(* Stop *)
	IF xStop THEN
		(* init. FB vel / abs / rel *)
		xMoveVel:=FALSE;
		xMoveRel:=FALSE;
		xMoveAbs:=FALSE;
		xMoveModulo:=FALSE;
		xNewVelocity:=FALSE;
		xNewPosition:=FALSE;
		xStartTimerComm:=FALSE;
		xHoming:=FALSE;
		IF (iTmpFctNr <> 19) THEN
			xCalcAngleRefIndex:=FALSE;
		END_IF;
		(* flag oscillation off *)
		xOscillation:=FALSE;
		(* FB stop *)
		xStopAxisVelCtrlActive:=FALSE;
		IF (T_Axis.T_Config_Gen.iTyp <> 1) THEN
			fbAxisStop(	Execute:=TRUE,
						Deceleration:=T_Axis.T_CtrleSingle.lrDecceleration,
						Jerk:=T_Axis.T_CtrleSingle.lrJerk,
						Axis:=T_AxisRefIn);
		ELSE
			IF NOT(gxZAxisVelocityCtrlActive) THEN
				fbAxisStop(	Execute:=TRUE,
							Deceleration:=T_Axis.T_CtrleSingle.lrDecceleration,
							Jerk:=T_Axis.T_CtrleSingle.lrJerk,
							Axis:=T_AxisRefIn);
			ELSE
				xStopAxisVelCtrlActive:=TRUE;
			END_IF;
		END_IF;
		(* select bit not moving *)
		dwTmp:=T_Axis.T_LiveValue.dwState AND 16#4;
		IF NOT(xStopAxisVelCtrlActive) THEN
			IF (fbAxisStop.Done AND dwTmp = 16#4) OR fbAxisStop.Error THEN
				IF fbAxisStop.Error OR (NOT(xResetAxis) AND NOT(xResetAX5000Axis) AND NOT(xCalcAngleRefIndex) )THEN
					xResetAxis:=xCalcAngleRefIndex:=xResetAX5000Axis:=FALSE;
				(* confirm reset if error activ or if reset is not activ *)
					T_Axis.T_CtrleSingle.xDone:=fbAxisStop.Done;
					T_Axis.T_CtrleSingle.xErr:= fbAxisStop.Error;
					T_Axis.T_CtrleSingle.udiErrorID:=fbAxisStop.ErrorID;
					(* desactiv reset axis *)
					IF xResetAxis THEN xResetAxis:=FALSE; END_IF
					IF (T_Axis.T_Config_Gen.iTyp = 1) AND gxZFollowDistanceError THEN
						T_Axis.T_CtrleSingle.xDone:=FALSE;
						T_Axis.T_CtrleSingle.xErr:= TRUE;
						T_Axis.T_CtrleSingle.udiErrorID:=16#4550;	(* Schleppabstandsfehler *)
					END_IF;
				END_IF
				(* flag stop off *)
				xStop:=FALSE;
				tTimeCommLeft1:=TimerCommTimeLeft1.ET;
				xStartTimerComm1:=FALSE;
				(* reset flag busy *)
				T_Axis.T_CtrleSingle.xBusyNewPosAndVel:=FALSE;
				(* Init. Stop FB *)
				fbAxisStop(Execute:=FALSE, Axis:=T_AxisRefIn);
				IF xActiveFollowError AND NOT(fbAxisStop.Error) THEN
					T_Axis.T_CtrleSingle.xDone:=FALSE;
					T_Axis.T_CtrleSingle.xErr:= FALSE;
					T_Axis.T_CtrleSingle.udiErrorID:=0;
					xActiveFollowError:=FALSE;
					iStepResetFB:=1;
					xResetAxis:=TRUE;
					RETURN;
				END_IF;
				IF gxSpindleOverloadError AND (T_Axis.T_Config_Gen.iTyp = 2) THEN
					gxSpindleOverloadError:=FALSE;
					T_Axis.T_CtrleSingle.xDone:=FALSE;
					T_Axis.T_CtrleSingle.xErr:= TRUE;
					T_Axis.T_CtrleSingle.udiErrorID:=16#F502;
				END_IF;
			END_IF
		ELSE
			CASE iStopAxis OF
			1:	TONWaitStop(IN:=FALSE);
				iStepResetFB:=1;
				xResetAxis:=TRUE;
				iStopAxis:=iStopAxis + 1;
			2:	IF NOT(xResetAxis) THEN
					iStopAxis:=iStopAxis + 1;
				END_IF;
			3:	TONWaitStop(IN:=TRUE,PT:=T#0.3s);
				IF TONWaitStop.Q THEN
					TONWaitStop(IN:=FALSE);
					T_Axis.T_CtrleSingle.xDone:=TRUE;
					T_Axis.T_CtrleSingle.xErr:= FALSE;
					T_Axis.T_CtrleSingle.udiErrorID:=16#0;
					xStop:=FALSE;
					xStopAxisVelCtrlActive:=FALSE;
					iStopAxis:=1;
					IF (T_Axis.T_Config_Gen.iTyp = 1) AND gxZFollowDistanceError THEN
						T_Axis.T_CtrleSingle.xDone:=FALSE;
						T_Axis.T_CtrleSingle.xErr:= TRUE;
						T_Axis.T_CtrleSingle.udiErrorID:=16#4550;	(* Schleppabstandsfehler *)
					END_IF;
				END_IF;
			END_CASE;
		END_IF;
	ELSE fbAxisStop(Execute:=FALSE, Axis:=T_AxisRefIn); END_IF

(* Velocity *)
	IF xMoveVel AND NOT(fbAxisMoveVelocity.InVelocity) THEN
		IF T_Axis.T_CtrleSingle.lrVelocity >= 0 THEN
		(* positiv direction =1*)
			iDirectionVel:=MC_Positive_Direction;
		ELSE
		(* negativ direction =3*)
			iDirectionVel:=MC_Negative_Direction;
		END_IF
		IF (T_Axis.T_Config_Gen.iTyp <> 2) THEN
			rVelocity:=ABS(lrOverrideVel);
		ELSE
			rVelocity:=ABS(lrOverrideVel) * T_Axis.T_CtrleSingle.lrScaleFactor;
		END_IF;
		fbAxisMoveVelocity(	Execute:=TRUE,
							Velocity:=rVelocity,
							Acceleration:=T_Axis.T_CtrleSingle.lrAcceleration,
							Deceleration:=T_Axis.T_CtrleSingle.lrDecceleration,
							Jerk:=T_Axis.T_CtrleSingle.lrJerk,
							Direction:=iDirectionVel,
							Axis:=T_AxisRefIn);
		IF fbAxisMoveVelocity.InVelocity OR fbAxisMoveVelocity.Error THEN
			T_Axis.T_CtrleSingle.xDone:=fbAxisMoveVelocity.InVelocity;
			T_Axis.T_CtrleSingle.xErr:= fbAxisMoveVelocity.Error;
			T_Axis.T_CtrleSingle.udiErrorID:=fbAxisMoveVelocity.ErrorID;
			(* flag velocity off *)
			xMoveVel:=FALSE;
			(* Init. FB Move *)
			fbAxisMoveVelocity(Execute:=FALSE, Axis:=T_AxisRefIn);
		END_IF
	ELSE fbAxisMoveVelocity(Execute:=FALSE, Axis:=T_AxisRefIn); END_IF

(* Move absolute *)
	IF xMoveAbs THEN
		fbAxisMoveAbsolute(	Execute:=TRUE,
							Position:=T_Axis.T_CtrleSingle.lrPosition,
							Velocity:=ABS(lrOverrideVel),
							Acceleration:=T_Axis.T_CtrleSingle.lrAcceleration,
							Deceleration:=T_Axis.T_CtrleSingle.lrDecceleration,
							Jerk:=T_Axis.T_CtrleSingle.lrJerk,
							Axis:=T_AxisRefIn);
		IF fbAxisMoveAbsolute.Done OR fbAxisMoveAbsolute.Error THEN
			IF NOT(xCalcAngleRefIndex) OR fbAxisMoveAbsolute.Error THEN
				xCalcAngleRefIndex:=FALSE;
				IF NOT(T_Axis.T_CtrleSingle.xErr) THEN	(* xNewVelocity könnte einen Fehler generiert haben, aber diese Funktion ist noch aktiv und darf daher nicht überschrieben werden *)
					T_Axis.T_CtrleSingle.xDone:=fbAxisMoveAbsolute.Done;
					T_Axis.T_CtrleSingle.xErr:= fbAxisMoveAbsolute.Error;
					T_Axis.T_CtrleSingle.udiErrorID:=fbAxisMoveAbsolute.ErrorID;
				END_IF;
				(* test if move has been stopped *)
				IF fbAxisMoveAbsolute.ErrorID = 16#4B00 THEN
				(* clear error *)
					T_Axis.T_CtrleSingle.xDone:=TRUE;
					T_Axis.T_CtrleSingle.xErr:= FALSE;
					T_Axis.T_CtrleSingle.udiErrorID:=16#0;
				END_IF
			END_IF;
			(* flag move absolute off *)
			xMoveAbs:=FALSE;
			(* init. FB *)
			fbAxisMoveAbsolute(Execute:=FALSE, Axis:=T_AxisRefIn);
		END_IF
	ELSE fbAxisMoveAbsolute(Execute:=FALSE, Axis:=T_AxisRefIn); END_IF

(* Move relative *)
	IF xMoveRel THEN
		IF (T_Axis.T_Config_Gen.iTyp <> 2) THEN
			lrDistance:=T_Axis.T_CtrleSingle.lrDistance;
		ELSE
			CASE T_ExchgParam.bToolSpindleActive OF
			1:	(* Maxon Spindel *)
				lrDistance:=T_Axis.T_CtrleSingle.lrDistance / grScaleSAxis_Distance_SM;
			2,3:	(* Beckhoff Spindel *)
				lrDistance:=T_Axis.T_CtrleSingle.lrDistance / grScaleSAxis_Distance_L;
			END_CASE;
		END_IF;
		fbAxisMoveRelative(	Execute:=TRUE,
							Distance:=lrDistance,
							Velocity:=lrOverrideVel,
							Acceleration:=T_Axis.T_CtrleSingle.lrAcceleration,
							Deceleration:=T_Axis.T_CtrleSingle.lrDecceleration,
							Jerk:=T_Axis.T_CtrleSingle.lrJerk,
							Axis:=T_AxisRefIn);
		IF fbAxisMoveRelative.Done OR fbAxisMoveRelative.Error THEN
			IF (NOT(xOscillation) AND NOT(xCalcAngleRefIndex)) OR fbAxisMoveRelative.Error THEN
				xOscillation:=xCalcAngleRefIndex:=FALSE;
			(* normal control variable settings if oscillation disable *)
				IF NOT(T_Axis.T_CtrleSingle.xErr) THEN	(* xNewVelocity könnte einen Fehler generiert haben, aber diese Funktion ist noch aktiv und darf daher nicht überschrieben werden *)
					T_Axis.T_CtrleSingle.xDone:=fbAxisMoveRelative.Done;
					T_Axis.T_CtrleSingle.xErr:= fbAxisMoveRelative.Error;
					T_Axis.T_CtrleSingle.udiErrorID:=fbAxisMoveRelative.ErrorID;
				END_IF;
				(* test if move has been stopped *)
				IF fbAxisMoveRelative.ErrorID = 16#4B00 THEN
				(* clear error *)
					T_Axis.T_CtrleSingle.xDone:=TRUE;
					T_Axis.T_CtrleSingle.xErr:= FALSE;
					T_Axis.T_CtrleSingle.udiErrorID:=16#0;
				END_IF
			END_IF
			(* flag move relative off *)
			xMoveRel:=FALSE;
			(* init. FB *)
			fbAxisMoveRelative(Execute:=FALSE, Axis:=T_AxisRefIn);
		END_IF
	ELSE fbAxisMoveRelative(Execute:=FALSE, Axis:=T_AxisRefIn); END_IF

(* Move modulo *)
	IF xMoveModulo THEN
		fbAxisMoveModulo(	Execute:= TRUE,
							Position:= T_Axis.T_CtrleSingle.lrPosition,
							Velocity:= ABS(lrOverrideVel),
							Acceleration:= T_Axis.T_CtrleSingle.lrAcceleration,
							Deceleration:= T_Axis.T_CtrleSingle.lrDecceleration,
							Jerk:= T_Axis.T_CtrleSingle.lrJerk,
							Direction:= T_Axis.T_CtrleSingle.iModuloDirection,
							Axis:= T_AxisRefIn);
		IF fbAxisMoveModulo.Done OR fbAxisMoveModulo.Error THEN
			xCalcAngleRefIndex:=FALSE;
			T_Axis.T_CtrleSingle.xDone:=fbAxisMoveModulo.Done;
			T_Axis.T_CtrleSingle.xErr:= fbAxisMoveModulo.Error;
			T_Axis.T_CtrleSingle.udiErrorID:=fbAxisMoveModulo.ErrorID;
			(* test if move has been stopped *)
			IF fbAxisMoveModulo.ErrorID = 16#4B00 THEN
			(* clear error *)
				T_Axis.T_CtrleSingle.xDone:=TRUE;
				T_Axis.T_CtrleSingle.xErr:= FALSE;
				T_Axis.T_CtrleSingle.udiErrorID:=16#0;
			END_IF
			(* flag move absolute off *)
			xMoveModulo:=FALSE;
			(* init. FB *)
			fbAxisMoveModulo(Execute:=FALSE, Axis:=T_AxisRefIn);
		END_IF
	ELSE fbAxisMoveModulo(Execute:=FALSE, Axis:=T_AxisRefIn); END_IF

(* Homing *)
	IF xHoming THEN
		IF(T_Axis.T_Config_Gen.iTyp=1) THEN
			lrSetPosition:=T_Axis.T_CtrleSingle.rSetPosition + lrNullPointOffset;
		ELSE
			lrSetPosition:=T_Axis.T_CtrleSingle.rSetPosition;
		END_IF;
		fbAxisHoming(	Execute:=TRUE,
						Position:=lrSetPosition,
						bCalibrationCam:=xRefHoming,
						Axis:=T_AxisRefIn,
						AxisOut:=T_AxisRefOut);
		IF fbAxisHoming.Done OR fbAxisHoming.Error THEN
			IF NOT(xCalcAngleRefIndex) OR fbAxisHoming.Error THEN
				xCalcAngleRefIndex:=FALSE;
				T_Axis.T_CtrleSingle.xDone:=fbAxisHoming.Done;
				T_Axis.T_CtrleSingle.xErr:= fbAxisHoming.Error;
				T_Axis.T_CtrleSingle.udiErrorID:=fbAxisHoming.ErrorID;
			END_IF;
			(* flag homing off *)
			xHoming:=FALSE;
			(* Init. FB Homing *)
			fbAxisHoming(	Execute:=FALSE,
							Axis:=T_AxisRefIn,
							AxisOut:=T_AxisRefOut);
		END_IF
	ELSE
		fbAxisHoming(	Execute:=FALSE,
						Axis:=T_AxisRefIn,
						AxisOut:=T_AxisRefOut);
	END_IF

(* Set override *)
	IF xOverride THEN
		fbAxisSetOverride(Execute:=TRUE,
						Override:=T_Axis.T_CtrleSingle.dwOverride,
						AxisRefIn:=T_AxisRefIn,
						AxisRefOut:=T_AxisRefOut);
		IF fbAxisSetOverride.Done OR fbAxisSetOverride.Error THEN
			T_Axis.T_CtrleSingle.xDone:=fbAxisSetOverride.Done;
			T_Axis.T_CtrleSingle.xErr:= fbAxisSetOverride.Error;
			T_Axis.T_CtrleSingle.udiErrorID:=fbAxisSetOverride.ErrorID;
			(* flag override off *)
			xOverride:=FALSE;
			(* Init. FB Override *)
			fbAxisSetOverride(Execute:=FALSE,
							AxisRefIn:=T_AxisRefIn,
							AxisRefOut:=T_AxisRefOut);
		END_IF
	ELSE
		fbAxisSetOverride(Execute:=FALSE,
						AxisRefIn:=T_AxisRefIn,
						AxisRefOut:=T_AxisRefOut);
	END_IF

(* Set new position *)
	IF xSetPosition THEN
		fbAxisSetPosition(	Execute:=TRUE, Position:=T_Axis.T_CtrleSingle.rSetPosition, Axis:=T_AxisRefIn);
		IF fbAxisSetPosition.Done OR fbAxisSetPosition.Error THEN
			T_Axis.T_CtrleSingle.xDone:=fbAxisSetPosition.Done;
			T_Axis.T_CtrleSingle.xErr:= fbAxisSetPosition.Error;
			T_Axis.T_CtrleSingle.udiErrorID:=fbAxisSetPosition.ErrorID;
			(* flag set position off *)
			xSetPosition:=FALSE;
			(* Init. FB set position *)
			fbAxisSetPosition(Execute:=FALSE, Axis:=T_AxisRefIn);
		END_IF
	ELSE fbAxisSetPosition(Execute:=FALSE, Axis:=T_AxisRefIn); END_IF

(* set new velocity or new position *)
	IF xNewVelocity OR xNewPosition THEN
		IF (T_Axis.T_Config_Gen.iTyp <> 2) THEN
			rVelocity:=ABS(lrOverrideVel);
		ELSE
			rVelocity:=ABS(lrOverrideVel) * T_Axis.T_CtrleSingle.lrScaleFactor;
		END_IF;
		IF NOT(xOscillation) OR xNewPosition THEN
			IF NOT(T_Axis.T_CtrleSingle.xNotMoving) THEN
				xNoHWError:=FALSE;
				IF xNewVelocity THEN
				(* new velocity *)
					fbAxisNewPosAndVel(	Execute:=TRUE,
										Mode:=2,
										NewVelo:=ABS(rVelocity),
										Axis:=T_AxisRefIn);
				ELSE
				(* new position *)
					fbAxisNewPosAndVel(	Execute:=TRUE,
										Mode:=3,
										NewPos:=T_Axis.T_CtrleSingle.lrPosition,
										NewVelo:=lrOverrideVel,
										Axis:=T_AxisRefIn);
				END_IF
			ELSE
				xNoHWError:=TRUE;
			END_IF;
			IF fbAxisNewPosAndVel.Done OR fbAxisNewPosAndVel.Error OR xNoHWError THEN
			(* confirm end function *)
				IF xMovement THEN
					IF NOT(xNoHWError) THEN
						T_Axis.T_CtrleSingle.xDone:=FALSE;
					ELSE
						IF xMoveAbs OR xMoveRel OR xMoveModulo THEN
							T_Axis.T_CtrleSingle.xDone:=FALSE;
						ELSE
							T_Axis.T_CtrleSingle.xDone:=TRUE;
						END_IF;
					END_IF;
				ELSE
					IF NOT(xNoHWError) THEN
						T_Axis.T_CtrleSingle.xDone:=fbAxisNewPosAndVel.Done;
					ELSE
						T_Axis.T_CtrleSingle.xDone:=TRUE;
					END_IF;
				END_IF;
				IF NOT(xNoHWError) THEN
(*					IF (fbAxisNewPosAndVel.ErrorID <> 17022) AND (fbAxisNewPosAndVel.ErrorID <> 16900) THEN	(* Fehler 17022: Während Beschleunigungsphase wird eine neue Geschwindigkeit angefordert und erzeugt ein NC Fehler, Achse fährt aber Normal weiter, daher wird dieser Fehler nicht berücksichtigt *)
*)					IF NOT(xMovement) THEN
						T_Axis.T_CtrleSingle.xErr:= fbAxisNewPosAndVel.Error;
						T_Axis.T_CtrleSingle.udiErrorID:=fbAxisNewPosAndVel.ErrorID;
					END_IF;
					IF (fbAxisNewPosAndVel.ErrorID = 17022) THEN
						diStepErrorCounter:=diStepErrorCounter + 1;
					END_IF;
					IF (fbAxisNewPosAndVel.ErrorID = 16900) THEN
						diStepErrorCounter1:=diStepErrorCounter1 + 1;
					END_IF;
				ELSE
					xNoHWError:=FALSE;
					T_Axis.T_CtrleSingle.xErr:= FALSE;
					T_Axis.T_CtrleSingle.udiErrorID:=0;
				END_IF;
				(* flag new velocity off and new position off *)
				xNewVelocity:=FALSE;
				xNewPosition:=FALSE;
				T_Axis.T_CtrleSingle.iFunction:=iTmpFctNr;
				(* Init. flag busy *)
				T_Axis.T_CtrleSingle.xBusyNewPosAndVel:=FALSE;
				(* Init. FB New pos and vel *)
				fbAxisNewPosAndVel(	Execute:=FALSE, Axis:=T_AxisRefIn);
				tTimeCommLeft:=TimerCommTimeLeft.ET;
				xStartTimerComm:=FALSE;
			END_IF
		ELSE
			(* velocity calculation *)
			IF T_Axis.T_Oscillation.rFrequence >= 0 AND T_Axis.T_Oscillation.rFrequence <= 1 THEN
				rTmpFrequence:=1.05 * T_Axis.T_Oscillation.rFrequence; END_IF
			IF T_Axis.T_Oscillation.rFrequence >=1 AND T_Axis.T_Oscillation.rFrequence <= 2 THEN
				rTmpFrequence:=1.25 * T_Axis.T_Oscillation.rFrequence; END_IF
			IF T_Axis.T_Oscillation.rFrequence >= 2 AND T_Axis.T_Oscillation.rFrequence <= 3 THEN
				rTmpFrequence:=2.5 * T_Axis.T_Oscillation.rFrequence; END_IF
			IF T_Axis.T_Oscillation.rFrequence >= 3 AND T_Axis.T_Oscillation.rFrequence <= 4 THEN
				rTmpFrequence:=5 * T_Axis.T_Oscillation.rFrequence; END_IF
			IF T_Axis.T_Oscillation.rFrequence >= 4 AND T_Axis.T_Oscillation.rFrequence <= 5 THEN
				rTmpFrequence:=10 * T_Axis.T_Oscillation.rFrequence; END_IF
			IF T_Axis.T_Oscillation.rFrequence > 5 THEN rTmpFrequence:=20; END_IF
			lrTmpVelocity:=(rTmpFrequence * 2 + 1 / rTmpFrequence) * ABS(T_Axis.T_Oscillation.rOffset);
			IF lrTmpVelocity > 250 THEN T_Axis.T_CtrleSingle.lrVelocity:=250;
				ELSE T_Axis.T_CtrleSingle.lrVelocity:=lrTmpVelocity; END_IF
			IF xMovement THEN
				T_Axis.T_CtrleSingle.xDone:=FALSE;
			ELSE
				T_Axis.T_CtrleSingle.xDone:=TRUE;
			END_IF;
			T_Axis.T_CtrleSingle.xErr:= FALSE;
			T_Axis.T_CtrleSingle.udiErrorID:=0;
			xNewVelocity:=FALSE;
			T_Axis.T_CtrleSingle.iFunction:=iTmpFctNr;
			T_Axis.T_CtrleSingle.xBusyNewPosAndVel:=FALSE;
			tTimeCommLeft:=TimerCommTimeLeft.ET;
			xStartTimerComm:=FALSE;
		END_IF;
	ELSE IF NOT(xNewVelocity) AND NOT( xNewPosition) THEN fbAxisNewPosAndVel(Execute:=FALSE, Axis:=T_AxisRefIn); END_IF
	END_IF

(* Set or reset reference flag *)
	IF xSetReferenceFlag OR xResetReferenceFlag THEN
		IF xSetReferenceFlag THEN
		(* set reference flag *)
			xTmp:=TRUE;
		ELSE xTmp:=FALSE;
		END_IF
		fbAxisSetReferenceFlag(Execute:=TRUE, ReferenceFlag:=xTmp, Axis:=T_AxisRefIn);
		IF fbAxisSetReferenceFlag.Done OR fbAxisSetReferenceFlag.Error THEN
			T_Axis.T_CtrleSingle.xDone:=fbAxisSetReferenceFlag.Done;
			T_Axis.T_CtrleSingle.xErr:= fbAxisSetReferenceFlag.Error;
			T_Axis.T_CtrleSingle.udiErrorID:=fbAxisSetReferenceFlag.ErrorID;
			(* set flag 'reference flag' off *)
			xSetReferenceFlag:=FALSE;
			xResetReferenceFlag:=FALSE;
			(* Init. FB set reference *)
			fbAxisSetReferenceFlag(Execute:=FALSE, Axis:=T_AxisRefIn);
		END_IF
	ELSE fbAxisSetReferenceFlag(Execute:=FALSE, Axis:=T_AxisRefIn); END_IF

(* set/reset control position *)
	IF xCtrlePositionOn THEN
		fbExtSetPointGenEnable(	Execute:=TRUE,
								Axis:=T_AxisRefIn);
		IF fbExtSetPointGenEnable.Done OR fbExtSetPointGenEnable.Error THEN
			T_Axis.T_CtrleSingle.xDone:=fbExtSetPointGenEnable.Done;
			T_Axis.T_CtrleSingle.xErr:= fbExtSetPointGenEnable.Error;
			T_Axis.T_CtrleSingle.udiErrorID:=fbExtSetPointGenEnable.ErrorID;
			(* reset flag *)
			xCtrlePositionOn:=FALSE;
		END_IF
	ELSE
		fbExtSetPointGenEnable(	Execute:=FALSE,
								Axis:=T_AxisRefIn);
	END_IF
	IF xCtrlePositionOff THEN
		fbExtSetPointGenDisable(	Execute:=TRUE,
								Axis:=T_AxisRefIn);
		IF fbExtSetPointGenDisable.Done OR fbExtSetPointGenDisable.Error THEN
			T_Axis.T_CtrleSingle.xDone:=fbExtSetPointGenDisable.Done;
			T_Axis.T_CtrleSingle.xErr:= fbExtSetPointGenDisable.Error;
			T_Axis.T_CtrleSingle.udiErrorID:=fbExtSetPointGenDisable.ErrorID;
			(* reset flag *)
			xCtrlePositionOff:=FALSE;
		END_IF
	ELSE
		fbExtSetPointGenDisable(	Execute:=FALSE,
								Axis:=T_AxisRefIn);
	END_IF

(* calcultate angle between Reference Index and Reference Sensor *)
	IF xCalcAngleRefIndex THEN
		(* error or stop => stop oscillation *)
		IF T_Axis.T_CtrleSingle.xErr OR (xStop AND (iTmpFctNr <> 19)) THEN iStepOsc:=99; END_IF
		CASE iStepCalcRefIndex OF
		(* Drive referencing and search the Ref. Index *)
		1:	T_Axis.T_CtrleSingle.rSetPosition:=0.0;
			xHoming:=TRUE;
			iStepCalcRefIndex:=10;
			T_Axis.T_CtrleSingle.iZAngleRefIndex:=0;
			IF (T_Axis.T_Config_Gen.iTyp = 1) THEN
				lrTechUnitPerMotorTurn:=65536.0 * T_Axis.T_Config_ObjFileValue.lrScaleFactor;	(*65536 = inc pro Motorumdrehung-->so kann dann mit dem Skalierungsfaktor ermittelt werden, wieviel Tech.Einheit für eine Motorumdrehung*)
			ELSIF (T_Axis.T_Config_Gen.iTyp = 2) THEN
				lrTechUnitPerMotorTurn:=4096.0 * T_Axis.T_Config_ObjFileValue.lrScaleFactor;	(*4096 = inc pro Motorumdrehung-->so kann dann mit dem Skalierungsfaktor ermittelt werden, wieviel Tech.Einheit für eine Motorumdrehung*)
			ELSE
				lrTechUnitPerMotorTurn:=1048576.0 * T_Axis.T_Config_ObjFileValue.lrScaleFactor;	(*65536 = inc pro Motorumdrehung-->so kann dann mit dem Skalierungsfaktor ermittelt werden, wieviel Tech.Einheit für eine Motorumdrehung*)
			END_IF;
			IF lrTechUnitPerMotorTurn = 0.0 THEN
				IF (T_Axis.T_Config_Gen.iTyp = 1) THEN
					lrTechUnitPerMotorTurn:=2.5;	(* 2.5mm entsprechen einer Motorumdrehung für Stroke Achse *)
				END_IF;
				IF (T_Axis.T_Config_Gen.iTyp = 2) THEN
					lrTechUnitPerMotorTurn:=5.0 / 2.6;	(* 5mm = Steigung, 2.6 = Übersetzunh--<entsprechen einer Motorumdrehung für Z2 Achse *)
				END_IF;
				IF (T_Axis.T_Config_Gen.iTyp = 4) THEN
					lrTechUnitPerMotorTurn:=3.564;	(* 3.564 Grad entsprechen einer Motorumdrehung für PartDisc *)
				END_IF;
				IF (T_Axis.T_Config_Gen.iTyp = 5) THEN
					lrTechUnitPerMotorTurn:=18.0;	(* 18mm entsprechen einer Motorumdrehung für Shuttle *)
				END_IF;
			END_IF;
		10:	IF NOT(xHoming) THEN
				(* Go Absolut to the Reference Index *)
				T_Axis.T_CtrleSingle.lrPosition:=0.0;
				T_Axis.T_CtrleSingle.lrVelocity:=1.0;(*T_Axis.T_Config_ObjFileValue.lrCalVelocityBackward;*)
				T_Axis.T_CtrleSingle.lrAcceleration:=T_Axis.T_Config_ObjFileValue.lrAcceleration;
				T_Axis.T_CtrleSingle.lrDecceleration:=T_Axis.T_Config_ObjFileValue.lrDecceleration;
				T_Axis.T_CtrleSingle.lrJerk:=T_Axis.T_Config_ObjFileValue.lrJerk;
				dwOldOverride:=16#FFFF;
				xMoveAbs:=TRUE;
				iStepCalcRefIndex:=20;
			END_IF;
		20:	IF NOT(xMoveAbs) THEN
				(* Turn the Motor for 360 degrees relativ*)
				xCheckRefState:=xRefHoming;
				T_Axis.T_CtrleSingle.lrDistance:=lrTechUnitPerMotorTurn * -1.0;	(* Der eingesetzte Wert entscheidet ob links oder rechtsdrehend, daher ist es wichtig zu wissen dass der entsprechende Wert, Positiv oder Negativ, die Bewegung zum Ref.Sensor führt *)
				IF (T_Axis.T_Config_Gen.iTyp <> 4) THEN
					T_Axis.T_CtrleSingle.lrVelocity:=1.0;(*T_Axis.T_Config_ObjFileValue.lrCalVelocityBackward;*)
				ELSE
					T_Axis.T_CtrleSingle.lrVelocity:=0.1;(*T_Axis.T_Config_ObjFileValue.lrCalVelocityBackward;*)
				END_IF;
				T_Axis.T_CtrleSingle.lrAcceleration:=T_Axis.T_Config_ObjFileValue.lrAcceleration;
				T_Axis.T_CtrleSingle.lrDecceleration:=T_Axis.T_Config_ObjFileValue.lrDecceleration;
				T_Axis.T_CtrleSingle.lrJerk:=T_Axis.T_Config_ObjFileValue.lrJerk;
				dwOldOverride:=16#FFFF;
				xMoveRel:=TRUE;
				iStepCalcRefIndex:=30;
			END_IF;
		30:	IF (T_Axis.T_Config_Gen.iTyp <> 4) THEN
				T_Axis.T_CtrleSingle.iZAngleRefIndex:=ABS(LREAL_TO_INT((360.0 / lrTechUnitPerMotorTurn) * T_Axis.T_LiveValue.lrActualPosition));	(* Zeiger bewegt sich so dynamisch während der Fahrt auf der Suche des RefSensors *)
			ELSE
				T_Axis.T_CtrleSingle.iZAngleRefIndex:=ABS(LREAL_TO_INT((360.0 / lrTechUnitPerMotorTurn) * (360.0 - T_Axis.T_LiveValue.lrActualPosition)));	(* Zeiger bewegt sich so dynamisch während der Fahrt auf der Suche des RefSensors *)
			END_IF;
			IF xCheckRefState XOR xRefHoming THEN
				lrCapturePosition:=T_Axis.T_LiveValue.lrActualPosition;
				IF (ABS(lrCapturePosition) > ABS(lrTechUnitPerMotorTurn)) THEN
					lrCapturePosition:=360.0 - ABS(lrCapturePosition);
				END_IF;
				xStop:=TRUE;
				iStepCalcRefIndex:=40;
			END_IF;
			IF NOT(xMoveRel) AND NOT(xStop) THEN
				T_Axis.T_CtrleSingle.iZAngleRefIndex:=0;
				iStepCalcRefIndex:=50;
			END_IF;
		40:	IF NOT(xStop) THEN
				T_Axis.T_CtrleSingle.iZAngleRefIndex:=LREAL_TO_INT((360.0 / lrTechUnitPerMotorTurn) * lrCapturePosition);	(* Berechnung der Winkellage des RefIndex zum RefSensor *)
				IF (T_Axis.T_CtrleSingle.iZAngleRefIndex < 0) THEN
					T_Axis.T_CtrleSingle.iZAngleRefIndex:=T_Axis.T_CtrleSingle.iZAngleRefIndex * -1;
				END_IF;
				IF (T_Axis.T_CtrleSingle.iZAngleRefIndex > 360) THEN
					T_Axis.T_CtrleSingle.iZAngleRefIndex:=360;
				END_IF;
				iStepCalcRefIndex:=50;
			END_IF;
		(* End of calc of the ref index position *)
		50:	T_Axis.T_CtrleSingle.xDone:=TRUE;
			T_Axis.T_CtrleSingle.xErr:= FALSE;
			T_Axis.T_CtrleSingle.udiErrorID:=16#0;
			xCalcAngleRefIndex:=FALSE;
		END_CASE;
	ELSE
		iStepCalcRefIndex:=1;
	END_IF;

(* Oscillation *)
	IF xOscillation THEN
		(* error or stop => stop oscillation *)
		IF T_Axis.T_CtrleSingle.xErr OR xStop THEN iStepOsc:=99; END_IF
		CASE iStepOsc OF
		(* init. oscillation + start move*)
		1:	(* init. variable *)
			iOscCounter:=0;
			(* velocity calculation *)
			IF T_Axis.T_Oscillation.rFrequence >= 0 AND T_Axis.T_Oscillation.rFrequence <= 1 THEN
				rTmpFrequence:=1.05 * T_Axis.T_Oscillation.rFrequence; END_IF
			IF T_Axis.T_Oscillation.rFrequence >=1 AND T_Axis.T_Oscillation.rFrequence <= 2 THEN
				rTmpFrequence:=1.25 * T_Axis.T_Oscillation.rFrequence; END_IF
			IF T_Axis.T_Oscillation.rFrequence >= 2 AND T_Axis.T_Oscillation.rFrequence <= 3 THEN
				rTmpFrequence:=2.5 * T_Axis.T_Oscillation.rFrequence; END_IF
			IF T_Axis.T_Oscillation.rFrequence >= 3 AND T_Axis.T_Oscillation.rFrequence <= 4 THEN
				rTmpFrequence:=5 * T_Axis.T_Oscillation.rFrequence; END_IF
			IF T_Axis.T_Oscillation.rFrequence >= 4 AND T_Axis.T_Oscillation.rFrequence <= 5 THEN
				rTmpFrequence:=10 * T_Axis.T_Oscillation.rFrequence; END_IF
			IF T_Axis.T_Oscillation.rFrequence > 5 THEN rTmpFrequence:=20; END_IF
			lrTmpVelocity:=(rTmpFrequence * 2 + 1 / rTmpFrequence) * ABS(T_Axis.T_Oscillation.rOffset);
			IF lrTmpVelocity > 250 THEN T_Axis.T_CtrleSingle.lrVelocity:=250;
				ELSE T_Axis.T_CtrleSingle.lrVelocity:=lrTmpVelocity; END_IF
			(*
			(* velocity := frequence * (offset * 2) *)
			T_Axis.T_CtrleSingle.lrVelocity:=T_Axis.T_Oscillation.rFrequence * ABS(T_Axis.T_Oscillation.rOffset) * 2;
			*)
			(* set move *)
			T_Axis.T_CtrleSingle.lrDistance:=T_Axis.T_Oscillation.rOffset;
			xMoveRel:=TRUE;
			(* next step *)
			iStepOsc:=10;
		(* move *)
		10:	IF NOT(xMoveRel) THEN
				(* move *-1 *)
				T_Axis.T_CtrleSingle.lrDistance:=T_Axis.T_Oscillation.rOffset * -1;
				xMoveRel:=TRUE;
				(* next step *)
				iStepOsc:=20;
			END_IF
		(* osc +1 *)
		20:	IF NOT(xMoveRel) THEN
				iOscCounter:=iOscCounter+1;
				IF iOscCounter < T_Axis.T_Oscillation.iCycle THEN
				(* move *)
					T_Axis.T_CtrleSingle.lrDistance:=T_Axis.T_Oscillation.rOffset;
					xMoveRel:=TRUE;
					(* next step *)
					iStepOsc:=10;
				ELSE
				(* oscillation done *)
					T_Axis.T_CtrleSingle.xDone:=TRUE;
					T_Axis.T_CtrleSingle.xErr:= FALSE;
					T_Axis.T_CtrleSingle.udiErrorID:=16#0;
					(* init FB *)
					fbAxisMoveRelative(Execute:=FALSE, Axis:=T_AxisRefIn);
					(* reset flag *)
					xOscillation:=FALSE;
				END_IF
			END_IF
		(* end oscillation *)
		99:	xOscillation:=FALSE;
		END_CASE
	ELSE
	(* init. variable *)
		iStepOsc:=1;
	END_IF

(* Default parameter value *)
	IF xDefaultAxisParameter THEN
		fbDefaultAxisPara(xDefaultValue:=TRUE,T_Axis:=T_Axis);
		T_Axis.T_CtrleSingle.xDone:=TRUE;
		T_Axis.T_CtrleSingle.xErr:= FALSE;
		T_Axis.T_CtrleSingle.udiErrorID:=0;
		(* flag DefaultParameter off *)
		xDefaultAxisParameter:=FALSE;
	END_IF

(* Set/Reset SW Pos limit switch *)
	IF xSetSWPosLimitSwitch OR xResetSWPosLimitSwitch THEN
		CASE iStepSWLimitSwitch OF
		(* control flag *)
		1:	(* init. next step *)
			iStepSWLimitSwitch:=iStepSWLimitSwitch + 1;
			IF T_Axis.T_CtrleSingle.xPower THEN
			(* axis power on, control axis flag *)
				IF (T_AxisRefIn.nStateDWord AND 16#4) = 16#0 THEN
				(* axis is moving, activ error *)
					iStepSWLimitSwitch:=912;
				END_IF
				IF (T_AxisRefIn.nStateDWord AND 16#20) = 16#20 THEN
				(* axis is in slave mode, activ error *)
					iStepSWLimitSwitch:=913;
				END_IF
			END_IF
		2:	IF NOT (fbAdsWrite.BUSY )  THEN
			(* send axis parameter *)
				fbAdsWrite(WRITE:=FALSE);
				IF xSetSWPosLimitSwitch THEN
					lrData:=1;
				ELSE
					lrData:=0;
				END_IF;
				wTmp:=LREAL_TO_WORD(lrData);
				dwAdrVar:=ADR(wTmp);
				fbAdsWrite(	NETID:='',
							PORT:=501,
							IDXGRP:=16#5000 + T_Axis.T_Config_Gen.udiNC_TaskIdxGrp,
							IDXOFFS:=16#C,
							LEN:=16#2,
							SRCADDR:=dwAdrVar,
							WRITE:=TRUE,
							TMOUT:=T#2s);
			ELSE
				fbAdsWrite(WRITE:=FALSE);
			END_IF
			IF NOT(fbAdsWrite.BUSY) AND NOT(fbAdsWrite.ERR) THEN
			(* determin the next step *)
				iStepSWLimitSwitch:=998;
			END_IF
			IF fbAdsWrite.ERR THEN
			(* set next step  *)
				iStepSWLimitSwitch:=901;
			END_IF
				(* ads communication error *)
		901:	T_Axis.T_CtrleSingle.udiErrorID:=fbAdsWrite.ERRID;
			(* set next step *)
			iStepSWLimitSwitch:=991;
		(* error the axis is moving *)
		912:	T_Axis.T_CtrleSingle.udiErrorID:=16#F102;		(* Achsfunktion nicht ausführbar, da Achse in Bewegung ist *)
			(* set next step *)
			iStepSWLimitSwitch:=991;
		(* error the axis is in slave mode *)
		913:	T_Axis.T_CtrleSingle.udiErrorID:=16#F103;		(* Achsfunktion nicht ausführbar, da Achse in Slave Mode ist *)
			(* set next step *)
			iStepSWLimitSwitch:=991;
		(* set flag error *)
		991:	T_Axis.T_CtrleSingle.xDone:=FALSE;
			T_Axis.T_CtrleSingle.xErr:= TRUE;
			(* set last step *)
			iStepSWLimitSwitch:=999;
		(* set flag end function *)
		998:	T_Axis.T_CtrleSingle.xDone:=TRUE;
			T_Axis.T_CtrleSingle.xErr:= FALSE;
			T_Axis.T_CtrleSingle.udiErrorID:=0;
			(* set last step *)
			iStepSWLimitSwitch:=999;
		(* reset variable *)
		999:	xSetSWPosLimitSwitch:=xResetSWPosLimitSwitch:=FALSE;
		END_CASE
	ELSE
		IF NOT(xSendAxisParameter) THEN
			fbAdsWrite(WRITE:=FALSE);
		END_IF;
	END_IF

(* Send parameter *)
	IF xSendAxisParameter THEN
		CASE iStepSendPara OF
		(* control flag *)
		1:	(* init. next step *)
			iStepSendPara:=2;
			xSendBlock:=FALSE;
			IF T_Axis.T_CtrleSingle.xPower THEN
			(* axis power on, control axis flag *)
				IF (T_AxisRefIn.nStateDWord AND 16#4) = 16#0 THEN
				(* axis is moving, activ error *)
					iStepSendPara:=912;
				END_IF
				IF (T_AxisRefIn.nStateDWord AND 16#20) = 16#20 THEN
				(* axis is in slave mode, activ error *)
					iStepSendPara:=913;
				END_IF
			END_IF
		(* set power off *)
		2:	xRestoreAxisPower:=FALSE;
			IF T_Axis.T_CtrleSingle.xPower THEN
			(* set power off *)
				xPowerOff:=TRUE;
				xPowerOn:=NOT(xPowerOff);
				(* set flag restore *)
				xRestoreAxisPower:=TRUE;
				(* start time out *)
				TimerOutSendPara(IN:=FALSE);
				(* next step *)
				iStepSendPara:=3;
			ELSE
			(* already power off, activ send parameter *)
				iStepSendPara:=11;
			END_IF
		(* wait flag power off *)
		3:	IF NOT(T_Axis.T_CtrleSingle.xPower) THEN
			(* activ send parameter *)
				iStepSendPara:=11;
			END_IF
			IF TimerOutSendPara.Q THEN
			(* time out activ, set error *)
				iStepSendPara:=911;
			END_IF
		(* loop sending parameter *)
		11:	IF NOT (fbAdsWrite.BUSY )  AND NOT(xSendBlock) THEN
			(* send axis parameter *)
				fbAdsWrite(WRITE:=FALSE);
				CASE T_Axis.T_ParamFileObj[iPtrAxisParameter].udiLength OF
				(* True/False, 2 bytes*)
				2:	wTmp:=LREAL_TO_WORD(T_Axis.T_ParamFileObj[iPtrAxisParameter].lrReal);
					dwAdrVar:=ADR(wTmp);
				(* dword value, 4 bytes *)
				4:	dwTmp:=LREAL_TO_DWORD(T_Axis.T_ParamFileObj[iPtrAxisParameter].lrReal);
					dwAdrVar:=ADR(dwTmp);
				(* else, 8 bytes *)
				8:	dwAdrVar:=ADR(T_Axis.T_ParamFileObj[iPtrAxisParameter].lrReal);
				END_CASE
				fbAdsWrite(	NETID:='',
							PORT:=501,
							IDXGRP:=T_Axis.T_ParamFileObj[iPtrAxisParameter].udiIdxGroup,
							IDXOFFS:=T_Axis.T_ParamFileObj[iPtrAxisParameter].udiIndexOffset,
							LEN:=T_Axis.T_ParamFileObj[iPtrAxisParameter].udiLength,
							SRCADDR:=dwAdrVar,
							WRITE:=TRUE,
							TMOUT:=T#2s);
				(* next parameter *)
				iPtrAxisParameter:=iPtrAxisParameter+1;
				IF T_Axis.T_ParamFileObj[iPtrAxisParameter].udiIdxGroup = 0 THEN
				(* parameter list empty *)
					xSendBlock:=TRUE;
				END_IF
			ELSE
				fbAdsWrite(WRITE:=FALSE);
			END_IF
			IF NOT(fbAdsWrite.BUSY) AND NOT(fbAdsWrite.ERR) AND T_Axis.T_ParamFileObj[iPtrAxisParameter].udiIdxGroup = 0 THEN
			(* determin the next step *)
				IF xRestoreAxisPower THEN
				(* Restore axis power *)
					iStepSendPara:=101;
				ELSE
				(* set flag end function *)
					iStepSendPara:=998;
				END_IF
			END_IF
			IF fbAdsWrite.ERR THEN
			(* set next step  *)
				iStepSendPara:=901;
			END_IF
		(* set power on *)
		101:	xPowerOn:=TRUE;
			xPowerOff:=NOT(xPowerOn);
			(* start time out *)
			TimerOutSendPara(IN:=FALSE);
			(*  next step *)
			iStepSendPara:=102;
		(* wait flag power on *)
		102:	IF T_Axis.T_CtrleSingle.xPower THEN
			(* set flag end function *)
				iStepSendPara:=998;
			END_IF
			IF TimerOutSendPara.Q THEN
			(* time out activ, set error *)
				iStepSendPara:=911;
			END_IF
		(* ads communication error *)
		901:	T_Axis.T_CtrleSingle.udiErrorID:=fbAdsWrite.ERRID;
			(* set next step *)
			iStepSendPara:=991;
		(* time out after setting axis power on/off *)
		911:	T_Axis.T_CtrleSingle.udiErrorID:=16#F101;		(* Timeout beim senden der Achsparameter an NC Ebene *)
			(* set next step *)
			iStepSendPara:=991;
		(* error the axis is moving *)
		912:	T_Axis.T_CtrleSingle.udiErrorID:=16#F102;		(* Achsfunktion nicht ausführbar, da Achse in Bewegung ist *)
			(* set next step *)
			iStepSendPara:=991;
		(* error the axis is in slave mode *)
		913:	T_Axis.T_CtrleSingle.udiErrorID:=16#F103;		(* Achsfunktion nicht ausführbar, da Achse in Slave Mode ist *)
			(* set next step *)
			iStepSendPara:=991;
		(* set flag error *)
		991:	T_Axis.T_CtrleSingle.xDone:=FALSE;
			T_Axis.T_CtrleSingle.xErr:= TRUE;
			(* set last step *)
			iStepSendPara:=999;
		(* set flag end function *)
		998:	T_Axis.T_CtrleSingle.xDone:=TRUE;
			T_Axis.T_CtrleSingle.xErr:= FALSE;
			T_Axis.T_CtrleSingle.udiErrorID:=0;
			(* set last step *)
			iStepSendPara:=999;
		(* reset variable *)
		999:	xSendAxisParameter:=FALSE;
		END_CASE
	ELSE
		IF NOT(xSetSWPosLimitSwitch) AND NOT(xResetSWPosLimitSwitch) THEN
			fbAdsWrite(WRITE:=FALSE);
		END_IF;
	END_IF

(* send axis string *)
	IF xSendAxisString THEN
		(*IF NOT(fbADS_ReadWriteString.BUSY)   AND sReturnAxis = '' THEN
			fbADS_ReadWriteString(WRTRD:=FALSE);*)
			(* add carriage return and line feed *)
			sSendAxis:=CONCAT(T_Axis.T_CtrleSingle.sSend, '$R$L$00');
			fbADS_ReadWriteString(	NETID:=T_Axis.T_Config_Gen.sServoNetId,
									PORT:=200,
									IDXGRP:=1,
									IDXOFFS:=1,
									WRITELEN:=LEN(sSendAxis)-1,
									READLEN:=LEN(sReturnAxis)-1,
									SRCADDR:=ADR(sSendAxis),
									DESTADDR:=ADR(sReturnAxis),
									WRTRD:=TRUE,
									TMOUT:=T#3s);
		(*ELSE
			fbADS_ReadWriteString(WRTRD:=FALSE);
		END_IF*)
		IF NOT(fbADS_ReadWriteString.BUSY) AND NOT(fbADS_ReadWriteString.ERR) AND sReturnAxis <> '' THEN
			IF sSendAxis = sReturnAxis THEN
			(* received string correct *)
				T_Axis.T_CtrleSingle.xDone:=TRUE;
				T_Axis.T_CtrleSingle.xErr:= FALSE;
				T_Axis.T_CtrleSingle.udiErrorID:=0;
			ELSE
			(* received string incorrect, active error *)
				T_Axis.T_CtrleSingle.xDone:=FALSE;
				T_Axis.T_CtrleSingle.xErr:= TRUE;
				T_Axis.T_CtrleSingle.udiErrorID:=16#F106;		(* Falscher String empfangen beim senden von ASCII Zeichen an NC Ebene *)
			END_IF
			(* set flag xsendaxisstring off *)
			xSendAxisString:=FALSE;
		END_IF
		IF fbADS_ReadWriteString.ERR THEN
		(* set flag error *)
			T_Axis.T_CtrleSingle.xDone:=FALSE;
			T_Axis.T_CtrleSingle.xErr:= TRUE;
			T_Axis.T_CtrleSingle.udiErrorID:=fbADS_ReadWriteString.ERRID;
			(* set flag xsendaxisstring off *)
			xSendAxisString:=FALSE;
		END_IF
	ELSE
		fbADS_ReadWriteString(WRTRD:=FALSE);
	END_IF
END_FUNCTION_BLOCK

(* POU GENERAL/FBDefaultAxisValue, ST *)
FUNCTION_BLOCK FBDefaultAxisValue
VAR_INPUT
	xDefaultValue:BOOL:=FALSE;
	sDeviceName:STRING(255);
END_VAR
VAR_OUTPUT
END_VAR
VAR_IN_OUT
	T_Axis:ST_AXIS;
END_VAR
VAR
END_VAR
IF xDefaultValue THEN
	IF sDeviceName = 'Beckhoff' THEN
		CASE T_Axis.T_Config_Gen.iTyp OF
		(* linear axis Bore 800 *)
		1:	T_Axis.T_FileObj.sData[1]:='01:idxGrp:=16#4000;idxOff:=16#27;LEN:=16#8;Value:=200.0';(* Max velocity *)
			T_Axis.T_FileObj.sData[2]:='02:idxGrp:=16#4000;idxOff:=16#6;Len:=16#8;Value:=20.0';(* Vel Ref forward *)
			T_Axis.T_FileObj.sData[3]:='03:idxGrp:=16#4000;idxOff:=16#7;LEN:=16#8;Value:=20.0';(* Vel Ref backward *)
			T_Axis.T_FileObj.sData[4]:='04:idxGrp:=16#4000;idxOff:=16#101;Len:=16#8;Value:=3800.0';(* Acc *)
			T_Axis.T_FileObj.sData[5]:='05:idxGrp:=16#4000;idxOff:=16#102;Len:=16#8;Value:=3800.0';(* Dec *)
			T_Axis.T_FileObj.sData[6]:='06:idxGrp:=16#4000;idxOff:=16#103;Len:=16#8;Value:=80222.0';(* Jerk *)
			T_Axis.T_FileObj.sData[7]:='07:idxGrp:=16#4000;idxOff:=16#A;Len:=16#8;Value:=200.0';(* Rapid traverse vel *)
			T_Axis.T_FileObj.sData[8]:='08:idxGrp:=16#5000;idxOff:=16#B;Len:=16#2;Value:=0';(* Enable min soft pos *)
			T_Axis.T_FileObj.sData[9]:='09:idxGrp:=16#5000;idxOff:=16#D;Len:=16#8;Value:=0';(* Min soft pos *)
			T_Axis.T_FileObj.sData[10]:='10:idxGrp:=16#5000;idxOff:=16#C;Len:=16#2;Value:=0';(* Enable max soft pos *)
			T_Axis.T_FileObj.sData[11]:='11:idxGrp:=16#5000;idxOff:=16#E;Len:=16#8;Value:=0';(* Max soft pos *)
			T_Axis.T_FileObj.sData[12]:='12:idxGrp:=16#6000;idxOff:=16#10;Len:=16#2;Value:=1';(* Enable pos lag *)
			T_Axis.T_FileObj.sData[13]:='13:idxGrp:=16#6000;idxOff:=16#12;Len:=16#8;Value:=10.0';(* Max Pos lag *)
			T_Axis.T_FileObj.sData[14]:='14:idxGrp:=16#5000;idxOff:=16#8;Len:=16#2;Value:=0';(* Invert Enc counting *)
			T_Axis.T_FileObj.sData[15]:='15:idxGrp:=16#5000;idxOff:=16#6;Len:=16#8;Value:=3.81e-5';(* Enc scaling factor *)
			T_Axis.T_FileObj.sData[16]:='16:idxGrp:=16#5000;idxOff:=16#9;Len:=16#8;Value:=1';(* Enc modulo factor *)
			T_Axis.T_FileObj.sData[17]:='17:idxGrp:=16#5000;idxOff:=16#101;Len:=16#2;Value:=1';(* Enc dir for ref search *)
			T_Axis.T_FileObj.sData[18]:='18:idxGrp:=16#5000;idxOff:=16#102;Len:=16#2;Value:=0';(* Enc dir for sync impuls*)
			T_Axis.T_FileObj.sData[19]:='19:idxGrp:=16#5000;idxOff:=16#103;Len:=16#8;Value:=0';(* Enc ref value *)
			T_Axis.T_FileObj.sData[20]:='20:idxGrp:=16#5000;idxOff:=16#106;Len:=16#2;Value:=0';(* Enc Ext sync impuls *)
			T_Axis.T_FileObj.sData[21]:='21:idxGrp:=16#5000;idxOff:=16#107;Len:=16#4;Value:=5';(* Enc ref sequence *)
			T_Axis.T_FileObj.sData[22]:='22:idxGrp:=16#7000;idxOff:=16#6;Len:=16#2;Value:=0';(* Driver invert polarity *)
			T_Axis.T_FileObj.sData[23]:='23:idxGrp:=16#7000;idxOff:=16#101;Len:=16#8;Value:=220';(* Driver Max Ref vel *)
			T_Axis.T_FileObj.sData[24]:='24:idxGrp:=16#7000;idxOff:=16#102;Len:=16#8;Value:=0.75';(* Driver output ration *)
			T_Axis.T_FileObj.sData[25]:='25:idxGrp:=16#6000;idxOff:=16#B;Len:=16#8;Value:=1';(* Ctrler pre-ctrl weighting *)
			T_Axis.T_FileObj.sData[26]:='26:idxGrp:=16#6000;idxOff:=16#102;LEN:=16#8;Value:=50';(* Ctrler Kv factor *)
			T_Axis.T_FileObj.sData[27]:='';
		(* spindle axis Bore800 master *)
		2:	T_Axis.T_FileObj.sData[1]:='01:idxGrp:=16#4000;idxOff:=16#27;LEN:=16#8;Value:=24000.0';(* Max velocity *)
			T_Axis.T_FileObj.sData[2]:='02:idxGrp:=16#4000;idxOff:=16#6;Len:=16#8;Value:=60.0';(* Vel Ref forward *)
			T_Axis.T_FileObj.sData[3]:='03:idxGrp:=16#4000;idxOff:=16#7;LEN:=16#8;Value:=60.0';(* Vel Ref backward *)
			T_Axis.T_FileObj.sData[4]:='04:idxGrp:=16#4000;idxOff:=16#101;Len:=16#8;Value:=42000.0';(* Acc *)
			T_Axis.T_FileObj.sData[5]:='05:idxGrp:=16#4000;idxOff:=16#102;Len:=16#8;Value:=42000.0';(* Dec *)
			T_Axis.T_FileObj.sData[6]:='06:idxGrp:=16#4000;idxOff:=16#103;Len:=16#8;Value:=98000.0';(* Jerk *)
			T_Axis.T_FileObj.sData[7]:='07:idxGrp:=16#4000;idxOff:=16#A;Len:=16#8;Value:=24000.0';(* Rapid traverse vel *)
			T_Axis.T_FileObj.sData[8]:='08:idxGrp:=16#5000;idxOff:=16#B;Len:=16#2;Value:=0';(* Enable min soft pos *)
			T_Axis.T_FileObj.sData[9]:='09:idxGrp:=16#5000;idxOff:=16#D;Len:=16#8;Value:=0';(* Min soft pos *)
			T_Axis.T_FileObj.sData[10]:='10:idxGrp:=16#5000;idxOff:=16#C;Len:=16#2;Value:=0';(* Enable max soft pos *)
			T_Axis.T_FileObj.sData[11]:='11:idxGrp:=16#5000;idxOff:=16#E;Len:=16#8;Value:=0';(* Max soft pos *)
			T_Axis.T_FileObj.sData[12]:='12:idxGrp:=16#6000;idxOff:=16#10;Len:=16#2;Value:=1';(* Enable pos lag *)
			T_Axis.T_FileObj.sData[13]:='13:idxGrp:=16#6000;idxOff:=16#12;Len:=16#8;Value:=90.0';(* Max Pos lag *)
			T_Axis.T_FileObj.sData[14]:='14:idxGrp:=16#5000;idxOff:=16#8;Len:=16#2;Value:=0';(* Invert Enc counting *)
			T_Axis.T_FileObj.sData[15]:='15:idxGrp:=16#5000;idxOff:=16#6;Len:=16#8;Value:=0.00549';(* Enc scaling factor *)
			T_Axis.T_FileObj.sData[16]:='16:idxGrp:=16#5000;idxOff:=16#9;Len:=16#8;Value:=360';(* Enc modulo factor *)
			T_Axis.T_FileObj.sData[17]:='17:idxGrp:=16#5000;idxOff:=16#101;Len:=16#2;Value:=1';(* Enc dir for ref search *)
			T_Axis.T_FileObj.sData[18]:='18:idxGrp:=16#5000;idxOff:=16#102;Len:=16#2;Value:=0';(* Enc dir for sync impuls*)
			T_Axis.T_FileObj.sData[19]:='19:idxGrp:=16#5000;idxOff:=16#103;Len:=16#8;Value:=0';(* Enc ref value *)
			T_Axis.T_FileObj.sData[20]:='20:idxGrp:=16#5000;idxOff:=16#106;Len:=16#2;Value:=0';(* Enc Ext sync impuls *)
			T_Axis.T_FileObj.sData[21]:='21:idxGrp:=16#5000;idxOff:=16#107;Len:=16#4;Value:=5';(* Enc ref sequence *)
			T_Axis.T_FileObj.sData[22]:='22:idxGrp:=16#7000;idxOff:=16#6;Len:=16#2;Value:=0';(* Driver invert polarity *)
			T_Axis.T_FileObj.sData[23]:='23:idxGrp:=16#7000;idxOff:=16#101;Len:=16#8;Value:=26000';(* Driver Max Ref vel *)
			T_Axis.T_FileObj.sData[24]:='24:idxGrp:=16#7000;idxOff:=16#102;Len:=16#8;Value:=1';(* Driver output ration *)
			T_Axis.T_FileObj.sData[25]:='25:idxGrp:=16#6000;idxOff:=16#B;Len:=16#8;Value:=1';(* Ctrler pre-ctrl weighting *)
			T_Axis.T_FileObj.sData[26]:='26:idxGrp:=16#6000;idxOff:=16#102;LEN:=16#8;Value:=0.5';(* Ctrler Kv factor *)
			T_Axis.T_FileObj.sData[27]:='';
		(* handling *)
		4:	T_Axis.T_FileObj.sData[1]:='01:idxGrp:=16#4000;idxOff:=16#27;LEN:=16#8;Value:=500.0';(* Max velocity *)
			T_Axis.T_FileObj.sData[2]:='02:idxGrp:=16#4000;idxOff:=16#6;Len:=16#8;Value:=20.0';(* Vel Ref forward *)
			T_Axis.T_FileObj.sData[3]:='03:idxGrp:=16#4000;idxOff:=16#7;LEN:=16#8;Value:=10.0';(* Vel Ref backward *)
			T_Axis.T_FileObj.sData[4]:='04:idxGrp:=16#4000;idxOff:=16#101;Len:=16#8;Value:=3800.0';(* Acc *)
			T_Axis.T_FileObj.sData[5]:='05:idxGrp:=16#4000;idxOff:=16#102;Len:=16#8;Value:=3800.0';(* Dec *)
			T_Axis.T_FileObj.sData[6]:='06:idxGrp:=16#4000;idxOff:=16#103;Len:=16#8;Value:=80222.0';(* Jerk *)
			T_Axis.T_FileObj.sData[7]:='07:idxGrp:=16#4000;idxOff:=16#A;Len:=16#8;Value:=500.0';(* Rapid traverse vel *)
			T_Axis.T_FileObj.sData[8]:='08:idxGrp:=16#5000;idxOff:=16#B;Len:=16#2;Value:=0';(* Enable min soft pos *)
			T_Axis.T_FileObj.sData[9]:='09:idxGrp:=16#5000;idxOff:=16#D;Len:=16#8;Value:=0';(* Min soft pos *)
			T_Axis.T_FileObj.sData[10]:='10:idxGrp:=16#5000;idxOff:=16#C;Len:=16#2;Value:=0';(* Enable max soft pos *)
			T_Axis.T_FileObj.sData[11]:='11:idxGrp:=16#5000;idxOff:=16#E;Len:=16#8;Value:=0';(* Max soft pos *)
			T_Axis.T_FileObj.sData[12]:='12:idxGrp:=16#6000;idxOff:=16#10;Len:=16#2;Value:=1';(* Enable pos lag *)
			T_Axis.T_FileObj.sData[13]:='13:idxGrp:=16#6000;idxOff:=16#12;Len:=16#8;Value:=200.0';(* Max Pos lag *)
			T_Axis.T_FileObj.sData[14]:='14:idxGrp:=16#5000;idxOff:=16#8;Len:=16#2;Value:=1';(* Invert Enc counting *)
			T_Axis.T_FileObj.sData[15]:='15:idxGrp:=16#5000;idxOff:=16#6;Len:=16#8;Value:=3.433279926e-4';(* Enc scaling factor *)
			T_Axis.T_FileObj.sData[16]:='16:idxGrp:=16#5000;idxOff:=16#9;Len:=16#8;Value:=360';(* Enc modulo factor *)
			T_Axis.T_FileObj.sData[17]:='17:idxGrp:=16#5000;idxOff:=16#101;Len:=16#2;Value:=1';(* Enc dir for ref search *)
			T_Axis.T_FileObj.sData[18]:='18:idxGrp:=16#5000;idxOff:=16#102;Len:=16#2;Value:=0';(* Enc dir for sync impuls*)
			T_Axis.T_FileObj.sData[19]:='19:idxGrp:=16#5000;idxOff:=16#103;Len:=16#8;Value:=0';(* Enc ref value *)
			T_Axis.T_FileObj.sData[20]:='20:idxGrp:=16#5000;idxOff:=16#106;Len:=16#2;Value:=0';(* Enc Ext sync impuls *)
			T_Axis.T_FileObj.sData[21]:='21:idxGrp:=16#5000;idxOff:=16#107;Len:=16#4;Value:=5';(* Enc ref sequence *)
			T_Axis.T_FileObj.sData[22]:='22:idxGrp:=16#7000;idxOff:=16#6;Len:=16#2;Value:=1';(* Driver invert polarity *)
			T_Axis.T_FileObj.sData[23]:='23:idxGrp:=16#7000;idxOff:=16#101;Len:=16#8;Value:=550';(* Driver Max Ref vel *)
			T_Axis.T_FileObj.sData[24]:='24:idxGrp:=16#7000;idxOff:=16#102;Len:=16#8;Value:=0.1';(* Driver output ration *)
			T_Axis.T_FileObj.sData[25]:='25:idxGrp:=16#6000;idxOff:=16#B;Len:=16#8;Value:=1';(* Ctrler pre-ctrl weighting *)
			T_Axis.T_FileObj.sData[26]:='26:idxGrp:=16#6000;idxOff:=16#102;LEN:=16#8;Value:=120';(* Ctrler Kv factor *)
			T_Axis.T_FileObj.sData[27]:='';
		END_CASE
	END_IF
	IF sDeviceName = 'Maxon' THEN
		CASE T_Axis.T_Config_Gen.iTyp OF
		(* Spindel Master *)
		2:	T_Axis.T_FileObj.sData[1]:='01:idxGrp:=16#6402;idxOff:=16#0;LEN:=16#2;Value:=10';(* Motor typ *)
			T_Axis.T_FileObj.sData[2]:='02:idxGrp:=16#6410;idxOff:=16#1;Len:=16#2;Value:=668';(* Continuous current limit *)
			T_Axis.T_FileObj.sData[3]:='03:idxGrp:=16#6410;idxOff:=16#2;Len:=16#2;Value:=1336';(* Output current limit *)
			T_Axis.T_FileObj.sData[4]:='04:idxGrp:=16#607F;idxOff:=16#0;LEN:=16#4;Value:=18000';(* Max profile velocity *)
			T_Axis.T_FileObj.sData[5]:='05:idxGrp:=16#6083;idxOff:=16#0;LEN:=16#4;Value:=10000';(* Profile acceleration *)
			T_Axis.T_FileObj.sData[6]:='06:idxGrp:=16#6084;idxOff:=16#0;LEN:=16#4;Value:=10000';(* Profile decceleration *)
			T_Axis.T_FileObj.sData[7]:='07:idxGrp:=16#6085;idxOff:=16#0;Len:=16#4;Value:=10000';(* Profile quickstop *)
			T_Axis.T_FileObj.sData[8]:='08:idxGrp:=16#2210;idxOff:=16#1;Len:=16#2;Value:=128';(* Encoder pulse number *)
			T_Axis.T_FileObj.sData[9]:='09:idxGrp:=16#60F6;idxOff:=16#1;Len:=16#2;Value:=1301';(* Current Regulator P-Gain *)
			T_Axis.T_FileObj.sData[10]:='10:idxGrp:=16#60F6;idxOff:=16#2;Len:=16#2;Value:=898';(* Current Regulator I-Gain *)
			T_Axis.T_FileObj.sData[11]:='11:idxGrp:=16#60F9;idxOff:=16#1;Len:=16#2;Value:=2186';(* Speed Regulator P-Gain *)
			T_Axis.T_FileObj.sData[12]:='12:idxGrp:=16#60F9;idxOff:=16#2;Len:=16#2;Value:=555';(* Speed Regulator P-Gain *)
			T_Axis.T_FileObj.sData[13]:='13:idxGrp:=16#6065;idxOff:=16#0;Len:=16#4;Value:=2000';(* Max Following error *)
			T_Axis.T_FileObj.sData[14]:='14:idxGrp:=16#2300;idxOff:=16#2;LEN:=16#2;Value:=1';(* Scaling numerator *)
			T_Axis.T_FileObj.sData[15]:='14:idxGrp:=16#2300;idxOff:=16#3;LEN:=16#2;Value:=1';(* Scaling denominator *)
			T_Axis.T_FileObj.sData[16]:='14:idxGrp:=16#2300;idxOff:=16#4;LEN:=16#1;Value:=0';(* Digital position polarity *)
			T_Axis.T_FileObj.sData[17]:='';
		(* Spindel Slave *)
		3:	T_Axis.T_FileObj.sData[1]:='01:idxGrp:=16#6402;idxOff:=16#0;LEN:=16#2;Value:=10';(* Motor typ *)
			T_Axis.T_FileObj.sData[2]:='02:idxGrp:=16#6410;idxOff:=16#1;Len:=16#2;Value:=668';(* Continuous current limit *)
			T_Axis.T_FileObj.sData[3]:='03:idxGrp:=16#6410;idxOff:=16#2;Len:=16#2;Value:=1336';(* Output current limit *)
			T_Axis.T_FileObj.sData[4]:='04:idxGrp:=16#607F;idxOff:=16#0;LEN:=16#4;Value:=18000';(* Max profile velocity *)
			T_Axis.T_FileObj.sData[5]:='05:idxGrp:=16#6083;idxOff:=16#0;LEN:=16#4;Value:=10000';(* Profile acceleration *)
			T_Axis.T_FileObj.sData[6]:='06:idxGrp:=16#6084;idxOff:=16#0;LEN:=16#4;Value:=10000';(* Profile decceleration *)
			T_Axis.T_FileObj.sData[7]:='07:idxGrp:=16#6085;idxOff:=16#0;Len:=16#4;Value:=10000';(* Profile quickstop *)
			T_Axis.T_FileObj.sData[8]:='08:idxGrp:=16#2210;idxOff:=16#1;Len:=16#2;Value:=128';(* Encoder pulse number *)
			T_Axis.T_FileObj.sData[9]:='09:idxGrp:=16#60F6;idxOff:=16#1;Len:=16#2;Value:=1301';(* Current Regulator P-Gain *)
			T_Axis.T_FileObj.sData[10]:='10:idxGrp:=16#60F6;idxOff:=16#2;Len:=16#2;Value:=898';(* Current Regulator I-Gain *)
			T_Axis.T_FileObj.sData[11]:='11:idxGrp:=16#60F9;idxOff:=16#1;Len:=16#2;Value:=2186';(* Speed Regulator P-Gain *)
			T_Axis.T_FileObj.sData[12]:='12:idxGrp:=16#60F9;idxOff:=16#2;Len:=16#2;Value:=555';(* Speed Regulator P-Gain *)
			T_Axis.T_FileObj.sData[13]:='13:idxGrp:=16#6065;idxOff:=16#0;Len:=16#4;Value:=2000';(* Max Following error *)
			T_Axis.T_FileObj.sData[14]:='14:idxGrp:=16#2300;idxOff:=16#2;LEN:=16#2;Value:=1';(* Scaling numerator *)
			T_Axis.T_FileObj.sData[15]:='14:idxGrp:=16#2300;idxOff:=16#3;LEN:=16#2;Value:=1';(* Scaling denominator *)
			T_Axis.T_FileObj.sData[16]:='14:idxGrp:=16#2300;idxOff:=16#4;LEN:=16#1;Value:=1';(* Digital position polarity *)
			T_Axis.T_FileObj.sData[17]:='';
		END_CASE
	END_IF
END_IF
END_FUNCTION_BLOCK

(* POU FB_HARDWARE/FBHW_AXIS_LIVEVALUES, ST *)
FUNCTION_BLOCK FBHW_AXIS_LIVEVALUES
VAR_INPUT
	uiActualTorque: UINT;
	IiActualTorque: INT;	(* Drehmoment von AX5xxx Servo *)
	arxDigitalInput: ARRAY[1..8] OF BOOL;
END_VAR
VAR_OUTPUT
END_VAR
VAR_IN_OUT
	T_Axis:ST_AXIS;
	T_AxisRefIn:NCTOPLC_AXLESTRUCT;
END_VAR
VAR
	i:INT;
END_VAR
(* return actual axis state *)
T_Axis.T_LiveValue.dwState:=T_AxisRefIn.nStateDWord;
(* return actual torque value *)
IF NOT(T_Axis.T_CtrleSingle.xAX5000Active) THEN
	T_Axis.T_LiveValue.uiActualTorque:=uiActualTorque;
	IF T_Axis.T_LiveValue.uiActualTorque > 16#7FFF THEN
		(* negativ value *)
		T_Axis.T_LiveValue.diActualTorqueCalc:=UINT_TO_DINT(T_Axis.T_LiveValue.uiActualTorque) - 65535;
	ELSE
		(* positiv value *)
		T_Axis.T_LiveValue.diActualTorqueCalc:=UINT_TO_DINT(T_Axis.T_LiveValue.uiActualTorque);
	END_IF
ELSE
	T_Axis.T_LiveValue.diActualTorqueCalc:=IiActualTorque;
END_IF;
(* return actual velocity *)
IF (T_Axis.T_Config_Gen.iTyp <> 2) THEN
	T_Axis.T_LiveValue.lrActualVelocity:=T_AxisRefIn.fVeloIst;
ELSE
	CASE T_ExchgParam.bToolSpindleActive OF
	1:	(* Maxon Spindel *)
		IF (T_NovRam.T_Parameter.T_StationWork[gciStationSt1].T_TorqueSystem.rGearRatioGearBox <> 0.0) THEN
			T_Axis.T_LiveValue.lrActualVelocity:=T_AxisRefIn.fVeloIst/T_NovRam.T_Parameter.T_StationWork[gciStationSt1].T_TorqueSystem.rGearRatioGearBox;
		ELSE
			T_Axis.T_LiveValue.lrActualVelocity:=T_AxisRefIn.fVeloIst;
		END_IF;
	2,3:	(* Beckhoff Spindel L *)
		T_Axis.T_LiveValue.lrActualVelocity:=T_AxisRefIn.fVeloIst / T_Axis.T_CtrleSingle.lrScaleFactor;
	END_CASE;
END_IF;
(* return actual position *)
IF (T_Axis.T_Config_Gen.iTyp = 2) THEN
(* modulo position for rotativ axis*)
	CASE T_ExchgParam.bToolSpindleActive OF
	1:	(* Maxon Spindel *)
		T_Axis.T_LiveValue.lrActualPosition:=DINT_TO_REAL(REAL_TO_DINT(100.0 * T_AxisRefIn.fModuloPosIst * grScaleSAxis_Distance_SM) MOD 36000) / 100.0;
		T_Axis.T_LiveValue.lrActualPositionNotModulo:=DINT_TO_REAL(REAL_TO_DINT(100.0 * T_AxisRefIn.fPosIst * grScaleSAxis_Distance_SM) MOD 36000) / 100.0;
	2,3:	(* Beckhoff Spindel *)
		T_Axis.T_LiveValue.lrActualPosition:=DINT_TO_REAL(REAL_TO_DINT(100.0 * T_AxisRefIn.fModuloPosIst * grScaleSAxis_Distance_L) MOD 36000) / 100.0;
		T_Axis.T_LiveValue.lrActualPositionNotModulo:=DINT_TO_REAL(REAL_TO_DINT(100.0 * T_AxisRefIn.fPosIst * grScaleSAxis_Distance_L) MOD 36000) / 100.0;
	END_CASE;
ELSE
(* counter value *)
	T_Axis.T_LiveValue.lrActualPosition:=T_AxisRefIn.fPosIst;
END_IF
T_Axis.T_LiveValue.lrSollPosition:=T_AxisRefIn.fPosSoll;
(* return actual position *)
(*T_Axis.T_LiveValue.lrActualPosition:=T_AxisRefIn.fPosIst;*)
(* return the actual digital input state *)
T_Axis.T_LiveValue.bDigitalInput:=0;
FOR i := 0 TO 7 DO
	IF arxDigitalInput[i+1] THEN
		T_Axis.T_LiveValue.bDigitalInput:=T_Axis.T_LiveValue.bDigitalInput + MUX(i,1,2,4,8,16,32,64,128);
	END_IF
END_FOR;
END_FUNCTION_BLOCK

(* POU FB_HARDWARE/FBHW_AXIS_DC, ST *)
FUNCTION_BLOCK FBHW_AXIS_DC
VAR_INPUT
END_VAR
VAR_IN_OUT
	T_Axis_DC : ST_DC_AXIS;
	usiStatusWord : USINT;
	usiControlWord : USINT;
	iDataOut : INT;
	iDataIn : INT;
	T_HDD:ST_HDD;
END_VAR
VAR_OUTPUT
END_VAR
VAR
(* trigger *)
	RisingEdgeResetFB:R_TRIG;
	RisingEdgeExecute:R_TRIG;
	RisingEdgePowerOn:R_TRIG;
	RisingEdgePowerOff:R_TRIG;

(* variable *)
	xConfirmResetFB:BOOL:=FALSE;
	xResetAxis:BOOL:=FALSE;
	xReadFile:BOOL:=FALSE;
	xPowerOn:BOOL:=FALSE;
	xPowerOff:BOOL:=FALSE;
	xMoveVel:BOOL:=FALSE;
	xStop:BOOL:=FALSE;
	xSendAxisParameter:BOOL:=FALSE;
	xWriteRegister: BOOL:=FALSE;
	xReadRegister: BOOL:=FALSE;

	iStepPowerOnFB:INT:=0;
	iStepPowerOffFB:INT:=0;
	iStepReadFile:INT:=0;
	iStepResetFB:INT:=0;
	iStepStopFB:INT:=0;
	iStepMoveVelFB:INT:=0;
	iStepSendAxisParameterFB:INT:=0;
	iStepWriteRegister: INT;
	iStepReadRegister: INT;
	iTmpFctNr:INT:=0;

	diTimeCounter: DINT;
	diTmpTimeCounter:DINT;
	iIncVelocity:INT;

	TONAccelerator:TON;
	lrScaleFactor:LREAL:=346.64;
	lrInitFactor:LREAL:=1500.0;
	lrVelocity:LREAL;
	xTmpPowerOn: BOOL;
	xTmpPowerOff: BOOL;
	xTmpError: BOOL;
	iTmpDataOut: INT;
	xInitAxis: BOOL;
(* timer *)
	TimerOutSendPara:TON;
	TimerFileLocked:TON;
	TimerTimeOutFunction:TON;

	sDeleteData: ARRAY[1..csiMaxAxisFileObj] OF STRING(80);
	sTmp:STRING(255);
	i:INT:=0;
	fb_ConvertParaAxis:FBConvertParaAxis;
	T_AxisDummy:ST_AXIS;

	iPtrAxisParameter:INT:=1;
	wDataToSend:WORD:=0;
	xInitAxisActiv: BOOL;
	lrActualVelocity:LREAL:=0.0;
	TONWaitStop: TON;
	xTmp: BOOL;
	RisingEdgeCheckStartFct: R_TRIG;
	xDeleteCtrl: BOOL;
END_VAR
(* reset block function *)
	RisingEdgeResetFB(CLK:=T_Axis_DC.T_CtrleDCAxis.xReset);
	IF RisingEdgeResetFB.Q THEN
	(* Init. block function *)
	(* Init. variable *)
		xResetAxis:=FALSE;
		TONAccelerator(IN:=FALSE);
		TimerTimeOutFunction(IN:=FALSE);
		TimerFileLocked(IN:=FALSE);
		TimerOutSendPara(IN:=FALSE);
		xTmpError:=FALSE;
		lrActualVelocity:=0.0;
		usiControlWord:=0;
		iDataOut:=0;
		xTmpError:=FALSE;
		xResetAxis:=xReadFile:=xTmpPowerOn:=xTmpPowerOff:=xStop:=xMoveVel:=xSendAxisParameter:=xWriteRegister:=xReadRegister:=FALSE;
	(* int. structure *)
		T_Axis_DC.T_CtrleDCAxis.iFunction:=0;
		T_Axis_DC.T_CtrleDCAxis.xDone:=FALSE;
		T_Axis_DC.T_CtrleDCAxis.xErr:=FALSE;
		T_Axis_DC.T_CtrleDCAxis.udiErrorID:=0;
		T_Axis_DC.T_CtrleDCAxis.xPower:=FALSE;
		T_Axis_DC.T_CtrleDCAxis.xReady:=FALSE;
		T_Axis_DC.T_CtrleDCAxis.xNotMoving:=TRUE;
		(* set flag done *)
		xConfirmResetFB:=TRUE;
		(* disable status flag *)
		T_Axis_DC.T_CtrleDCAxis.xDone:=FALSE;
		T_Axis_DC.T_CtrleDCAxis.xErr:=FALSE;
		T_Axis_DC.T_CtrleDCAxis.udiErrorID:=0;
		(* exit function bloc *)
		RETURN;
	ELSE
		IF xConfirmResetFB THEN
		(* confirm reset FB *)
			T_Axis_DC.T_CtrleDCAxis.xDone:=TRUE;
			T_Axis_DC.T_CtrleDCAxis.xErr:=FALSE;
			T_Axis_DC.T_CtrleDCAxis.udiErrorID:=0;
			(* reset variable *)
			xConfirmResetFB:=FALSE;
		END_IF
	END_IF

(* return axis state *)

(* Check Timeout for Function *)
xTmp:= xStop OR xResetAxis OR xTmpPowerOn OR xTmpPowerOff OR xReadFile OR xMoveVel OR xSendAxisParameter OR xWriteRegister OR xReadRegister;
IF TimerTimeOutFunction.Q AND xTmp THEN
	xResetAxis:=xReadFile:=xTmpPowerOn:=xTmpPowerOff:=xStop:=xMoveVel:=xSendAxisParameter:=xWriteRegister:=xReadRegister:=FALSE;
	usiControlWord:=2#0;
	iDataOut:=2#0;
	T_Axis_DC.T_CtrleDCAxis.xDone:=FALSE;
	T_Axis_DC.T_CtrleDCAxis.xErr:= TRUE;
	T_Axis_DC.T_CtrleDCAxis.udiErrorID:=16#F200;	(* Function Time Out *)
	RETURN;
END_IF;

(* Timer *)
	TimerOutSendPara(IN:=TRUE, PT:=T#10S);
	TimerFileLocked(IN:=TRUE, PT:=T#10S);
	TimerTimeOutFunction(IN:=TRUE,PT:=T#10S);

(* detection start *)
	RisingEdgeExecute(CLK:=T_Axis_DC.T_CtrleDCAxis.xExecute);
	IF RisingEdgeExecute.Q THEN
		IF xStop AND (T_Axis_DC.T_CtrleDCAxis.iFunction <> 1) THEN
		(* can not execute a function when 'Stop' activ, except 'Reset' *)
			T_Axis_DC.T_CtrleDCAxis.xDone:=FALSE;
			T_Axis_DC.T_CtrleDCAxis.xErr:=TRUE;
			T_Axis_DC.T_CtrleDCAxis.udiErrorID:=16#F100;
			RETURN;
		END_IF
		CASE T_Axis_DC.T_CtrleDCAxis.iFunction OF
		(* Reset *)
		1:	T_Axis_DC.T_CtrleDCAxis.xReady:=TRUE;
			T_Axis_DC.T_CtrleDCAxis.xPower:=FALSE;
			xPowerOn:=FALSE;
			xPowerOff:=TRUE;
			xResetAxis:=TRUE;
			iTmpFctNr:=1;
			iStepResetFB:=1;
		(* Init *)
		2:	xReadFile:=TRUE;
			iStepReadFile:=1;
			iTmpFctNr:=2;
			xInitAxisActiv:=TRUE;
		(* Power ON *)
		3:	IF NOT(xPowerOn) THEN
				xPowerOn:=TRUE;
				xPowerOff:=NOT(xPowerOn);
				xTmpPowerOn:=TRUE;
				iTmpFctNr:=3;
				iStepPowerOnFB:=1;
			ELSE
				T_Axis_DC.T_CtrleDCAxis.xDone:=TRUE;
				T_Axis_DC.T_CtrleDCAxis.xErr:= FALSE;
				T_Axis_DC.T_CtrleDCAxis.udiErrorID:=16#0;
				iTmpFctNr:=3;
				iStepPowerOnFB:=1;
				RETURN;
			END_IF;
		(* Power Off *)
		4:	IF xPowerOn THEN
				xPowerOff:=TRUE;
				xPowerOn:=NOT(xPowerOff);
				xTmpPowerOff:=TRUE;
				iTmpFctNr:=4;
				iStepPowerOffFB:=1;
			ELSE
				T_Axis_DC.T_CtrleDCAxis.xDone:=TRUE;
				T_Axis_DC.T_CtrleDCAxis.xErr:= FALSE;
				T_Axis_DC.T_CtrleDCAxis.udiErrorID:=16#0;
				iTmpFctNr:=4;
				iStepPowerOffFB:=1;
				RETURN;
			END_IF;
		(* Stop *)
		5: 	xStop:=TRUE;
			iTmpFctNr:=5;
			iStepStopFB:=1;
		(* Velocity *)
		6:	xMoveVel:=TRUE;
			iTmpFctNr:=6;
			iStepMoveVelFB:=1;
		(* Send Parameter *)
		21: 	xSendAxisParameter:=TRUE;
			iStepSendAxisParameterFB:=1;
			iPtrAxisParameter:=1;
			iTmpFctNr:=21;
		(* Write Register *)
		24:	xWriteRegister:=TRUE;
			iTmpFctNr:=24;
			iStepWriteRegister:=1;
		(* Read Register *)
		25:	xReadRegister:=TRUE;
			iTmpFctNr:=25;
			iStepReadRegister:=1;
		ELSE
		(* function not implemented *)
			T_Axis_DC.T_CtrleDCAxis.xDone:=FALSE;
			T_Axis_DC.T_CtrleDCAxis.xErr:=TRUE;
			T_Axis_DC.T_CtrleDCAxis.udiErrorID:=16#F000;
			(* Exit FB *)
			RETURN;
		END_CASE
		(* Init. variable *)
		T_Axis_DC.T_CtrleDCAxis.xDone:=FALSE;
		T_Axis_DC.T_CtrleDCAxis.xErr:=FALSE;
		T_Axis_DC.T_CtrleDCAxis.udiErrorID:=0;
		(* Exit FB *)
		(*RETURN;*)
	END_IF

(* detect error *)
	xTmp:= xStop OR xResetAxis OR xTmpPowerOn OR xTmpPowerOff OR xReadFile OR xMoveVel OR xSendAxisParameter OR xWriteRegister OR xReadRegister;
	IF NOT(xTmp) THEN
		T_Axis_DC.T_CtrleDCAxis.xErr:=GETBIT32(usiStatusWord,6);
	END_IF;
	xTmp:= xStop OR xTmpPowerOn OR xTmpPowerOff OR xReadFile OR xMoveVel OR xSendAxisParameter OR xWriteRegister OR xReadRegister;
	IF xDeleteCtrl THEN
		xDeleteCtrl:=FALSE;
		usiControlWord:=2#0;
		RETURN;
	END_IF;
	RisingEdgeCheckStartFct(CLK:=xTmp);
	IF RisingEdgeCheckStartFct.Q THEN
		IF GETBIT32(usiStatusWord,6) THEN
			usiControlWord:=2#01000000;
			xDeleteCtrl:=TRUE;
			RETURN;
		END_IF;
	END_IF;

(* Reset function *)
	IF xResetAxis THEN
		xReadFile:=xTmpPowerOn:=xTmpPowerOff:=xStop:=xMoveVel:=xSendAxisParameter:=xWriteRegister:=xReadRegister:=FALSE;
		CASE iStepResetFB OF
		1:	TimerTimeOutFunction(IN:=FALSE);
			usiControlWord:=2#0;
			iDataOut:=2#0;
			lrActualVelocity:=0.0;
			iStepResetFB:=10;
		10:	IF (usiStatusWord = 16#0) THEN
				usiControlWord:=2#01000000;
				iStepResetFB:=20;
			ELSE
				usiControlWord:=2#01000000;
				iStepResetFB:=20;
			END_IF;
		20:	IF (usiStatusWord = 16#0) THEN
				usiControlWord:=2#0;
				iStepResetFB:=900;
			END_IF;
		900:	(* confirm reset *)
			IF NOT(xWriteRegister) THEN
				T_Axis_DC.T_CtrleDCAxis.xDone:=TRUE;
				T_Axis_DC.T_CtrleDCAxis.xErr:= FALSE;
				T_Axis_DC.T_CtrleDCAxis.udiErrorID:=16#0;
			END_IF;
			T_Axis_DC.T_CtrleDCAxis.xNotMoving:=TRUE;
			(* init. variable *)
			xResetAxis:=FALSE;
		END_CASE;
	END_IF;

(* Initialisation function *)
	IF xReadFile THEN
		CASE iStepReadFile OF
		(* start timeout *)
		1:	TimerTimeOutFunction(IN:=FALSE);
			TimerFileLocked(IN:=FALSE);
			T_Axis_DC.T_FileObj.sData:=sDeleteData;
			(* next step *)
			iStepReadFile:=10;
		(* start read *)
		10:	IF T_HDD.T_Ctrle.xDone AND NOT(T_HDD.T_Ctrle.xLocked) THEN
			(* activ read axis nc parameter *)
				T_HDD.T_Ctrle.xExecute:=TRUE;
				T_HDD.T_Ctrle.xLocked :=TRUE;
				T_HDD.T_Ctrle.iFunction:=1;
				sTmp:=CONCAT(cssRootPLC,'Bore800\Axis\File\');
				sTmp:=CONCAT(sTmp, T_Axis_DC.T_Config_Gen.sDeviceFileName);
				T_HDD.T_File.sPathAndFileName:=CONCAT(sTmp,'.txt');
				(* next step *)
				iStepReadFile:=20;
			ELSE
			(* activ error if time out done, HDD not ready *)
				IF TimerFileLocked.Q THEN
					 iStepReadFile:=997;
				END_IF;
			END_IF;
		(* wait done or error *)
		20:	IF T_HDD.T_Ctrle.xDone OR T_HDD.T_Ctrle.xErr THEN
				IF T_HDD.T_Ctrle.xErr  THEN
				(* active step error *)
					iStepReadFile:=998;
					T_HDD.T_Ctrle.xLocked:=FALSE;
				ELSE
				(* next step, init convert value *)
					iStepReadFile:=30;
					(* copy data from file *)
					i:=1;
					WHILE T_HDD.T_Data.sData[i] <> '' AND i <=csiMaxAxisFileObj AND i <= csiMaxFileLine DO
						T_Axis_DC.T_FileObj.sData[i]:=T_HDD.T_Data.sData[i];
						i:=i+1;
					END_WHILE;
					(* erase last line +1 *)
					IF i < csiMaxAxisFileObj THEN T_Axis_DC.T_FileObj.sData[i+1]:=''; END_IF
				END_IF;
			END_IF;
		(* init. convert *)
		30:	fb_ConvertParaAxis(	xStart:=FALSE,
								iConversion:=1,
								T_Axis:=T_AxisDummy,
								T_Axis_DC:=T_Axis_DC);
			(* next step, convert value *)
			iStepReadFile:=40;
		(* convert value *)
		40:	fb_ConvertParaAxis(	xStart:=TRUE,
								iConversion:=1,
								sDeviceName:='MaxonDC',
								T_Axis:=T_AxisDummy,
								T_Axis_DC:=T_Axis_DC);
			IF fb_ConvertParaAxis.xDone OR fb_ConvertParaAxis.xError THEN
				IF fb_ConvertParaAxis.xError THEN
					fb_ConvertParaAxis(	xStart:=FALSE,
										iConversion:=1,
										T_Axis:=T_AxisDummy,
										T_Axis_DC:=T_Axis_DC);
					(* active step error *)
					iStepReadFile:=999;
				ELSE
					(* activ state read successfull *)
					iStepReadFile:=900;
				END_IF;
				T_HDD.T_Ctrle.xLocked:=FALSE;
			END_IF;
		(* confirm reset *)
		900:	T_Axis_DC.T_CtrleDCAxis.xDone:=TRUE;
			T_Axis_DC.T_CtrleDCAxis.xErr:= FALSE;
			T_Axis_DC.T_CtrleDCAxis.udiErrorID:=16#0;
			(* init. variable *)
			xReadFile:=FALSE;
		997:	(* Error stage *)
			T_HDD.T_Ctrle.xReset:=TRUE;
			T_Axis_DC.T_CtrleDCAxis.xDone:=FALSE;
			T_Axis_DC.T_CtrleDCAxis.xErr:= TRUE;
			T_Axis_DC.T_CtrleDCAxis.udiErrorID:=16#F300;	(* Reading Harddisk timeout *)
			xReadFile:=FALSE;
		998:	(* Error stage *)
			T_HDD.T_Ctrle.xReset:=TRUE;
			T_Axis_DC.T_CtrleDCAxis.xDone:=FALSE;
			T_Axis_DC.T_CtrleDCAxis.xErr:= TRUE;
			T_Axis_DC.T_CtrleDCAxis.udiErrorID:=16#F400;	(* File does not exist *)
			xReadFile:=FALSE;
		999:	(* Error stage *)
			T_HDD.T_Ctrle.xReset:=TRUE;
			T_Axis_DC.T_CtrleDCAxis.xDone:=FALSE;
			T_Axis_DC.T_CtrleDCAxis.xErr:= TRUE;
			T_Axis_DC.T_CtrleDCAxis.udiErrorID:=16#F500;	(* File conversion error *)
			xReadFile:=FALSE;
		END_CASE;
	END_IF;

(* Power function *)
	RisingEdgePowerOn(CLK:=xTmpPowerOn);
	RisingEdgePowerOff(CLK:=xTmpPowerOff);
	IF xTmpPowerOn THEN
		CASE iStepPowerOnFB OF
			1:	TimerTimeOutFunction(IN:=FALSE);
				xMoveVel:=FALSE;
				usiControlWord:=2#0;
				iDataOut:=0;
				lrActualVelocity:=0.0;
				iStepPowerOnFB:=10;
				T_Axis_DC.T_CtrleDCAxis.xPower:=TRUE;
			10:	usiControlWord:=2#00100000;
				iStepPowerOnFB:=20;
			20:	IF ((USINT_TO_WORD(usiStatusWord) AND 2#00010000) = 2#00010000) THEN
					iStepPowerOnFB:=900;
				END_IF;
			900:	(* confirm reset *)
			T_Axis_DC.T_CtrleDCAxis.xNotMoving:=TRUE;
			T_Axis_DC.T_CtrleDCAxis.xDone:=TRUE;
			T_Axis_DC.T_CtrleDCAxis.xErr:= FALSE;
			T_Axis_DC.T_CtrleDCAxis.udiErrorID:=16#0;
			xTmpPowerOn:=FALSE;
		END_CASE;
	END_IF;
	IF xTmpPowerOff THEN
		CASE iStepPowerOffFB OF
			1:	TimerTimeOutFunction(IN:=FALSE);
				xMoveVel:=FALSE;
				lrActualVelocity:=0.0;
				usiControlWord:=2#0;
				iDataOut:=0;
				iStepPowerOffFB:=10;
				T_Axis_DC.T_CtrleDCAxis.xPower:=FALSE;
			10:	IF (usiStatusWord = 2#0) THEN
					iStepPowerOffFB:=900;
				END_IF;
			900:	(* confirm reset *)
			T_Axis_DC.T_CtrleDCAxis.xNotMoving:=TRUE;
			T_Axis_DC.T_CtrleDCAxis.xDone:=TRUE;
			T_Axis_DC.T_CtrleDCAxis.xErr:= FALSE;
			T_Axis_DC.T_CtrleDCAxis.udiErrorID:=16#0;
			xTmpPowerOff:=FALSE;
		END_CASE;
	END_IF;


(* Stop *)
	IF xStop THEN
		CASE iStepStopFB OF
		1:	TimerTimeOutFunction(IN:=FALSE);
			TONWaitStop(IN:=FALSE);
			IF (T_Axis_DC.T_CtrleDCAxis.tDecceleration = T#0s) OR (lrActualVelocity = 0.0) THEN
				usiControlWord:=2#00100000;
				iDataOut:=0;
				iStepStopFB:=35;
			ELSE
				iStepStopFB:=20;
			END_IF;
			lrActualVelocity:=0.0;
			xMoveVel:=FALSE;
			IF (T_Axis_DC.T_CtrleDCAxis.lrVelocity >= 0) THEN lrInitFactor:=1500; END_IF;
			IF (T_Axis_DC.T_CtrleDCAxis.lrVelocity < 0) THEN lrInitFactor:=-1500; END_IF;
			lrVelocity:=(T_Axis_DC.T_CtrleDCAxis.lrVelocity * lrScaleFactor) + lrInitFactor;
			IF (lrVelocity > 32767) THEN lrVelocity:=32767; END_IF;
			IF (lrVelocity < -32768) THEN lrVelocity:=-32768; END_IF;
		20:	diTimeCounter:=REAL_TO_DINT(TIME_TO_REAL(T_Axis_DC.T_CtrleDCAxis.tDecceleration) / TIME_TO_REAL(T#10ms));
			diTmpTimeCounter:=0;
			iIncVelocity:=DINT_TO_INT(LREAL_TO_DINT(lrVelocity)/diTimeCounter);
			IF (iIncVelocity = 0) THEN
				IF (lrVelocity >= 0.0) THEN
					iIncVelocity:=-1;
				END_IF;
				IF (lrVelocity < 0.0) THEN
					iIncVelocity:=1;
				END_IF;
			ELSE
				iIncVelocity:=iIncVelocity * -1;
			END_IF;
			iStepStopFB:=30;
		30:	iDataOut:=iDataOut + iIncVelocity;
			diTmpTimeCounter:=diTmpTimeCounter + 1;
			IF (diTmpTimeCounter >= diTimeCounter) THEN
				iDataOut:=0;
				iStepStopFB:=40;
			END_IF;
			RETURN;
		35:	TONWaitStop(IN:=TRUE,PT:=T#200ms);
			IF TONWaitStop.Q THEN
				iStepStopFB:=40;
			END_IF;
		40:	usiControlWord:=2#0;
			iDataOut:=0;
			iStepStopFB:=900;
		900:	(* confirm reset *)
			T_Axis_DC.T_CtrleDCAxis.xNotMoving:=TRUE;
			T_Axis_DC.T_CtrleDCAxis.xDone:=TRUE;
			T_Axis_DC.T_CtrleDCAxis.xErr:= FALSE;
			T_Axis_DC.T_CtrleDCAxis.udiErrorID:=16#0;
			(* init. variable *)
			xStop:=FALSE;
		END_CASE;
	END_IF;

(* Velocity *)
	IF xMoveVel  THEN
		CASE iStepMoveVelFB OF
		1:	TimerTimeOutFunction(IN:=FALSE);
			usiControlWord:=2#0;
			iDataOut:=2#0;
			lrScaleFactor:=T_Axis_DC.T_Config_Gen.lrScaleFactor;
			lrInitFactor:=T_Axis_DC.T_Config_Gen.lrInitFactor;
			IF (T_Axis_DC.T_CtrleDCAxis.lrVelocity >= 0) THEN lrInitFactor:=lrInitFactor; END_IF;
			IF (T_Axis_DC.T_CtrleDCAxis.lrVelocity < 0) THEN lrInitFactor:=-lrInitFactor*-1; END_IF;
			lrVelocity:=(T_Axis_DC.T_CtrleDCAxis.lrVelocity * lrScaleFactor) + lrInitFactor;
			IF (lrVelocity > 32767) THEN lrVelocity:=32767; END_IF;
			IF (lrVelocity < -32768) THEN lrVelocity:=-32768; END_IF;
			lrActualVelocity:=lrVelocity;
			iStepMoveVelFB:=10;
		10:	IF (T_Axis_DC.T_CtrleDCAxis.tAcceleration = T#0s) THEN
				usiControlWord:=2#00100000;
				iDataOut:=LREAL_TO_INT(lrVelocity);
				iStepMoveVelFB:=900;
			ELSE
				usiControlWord:=2#00100000;
				iDataOut:=0;
				iStepMoveVelFB:=20;
			END_IF;
		20:	diTimeCounter:=REAL_TO_DINT(TIME_TO_REAL(T_Axis_DC.T_CtrleDCAxis.tAcceleration) / TIME_TO_REAL(T#10ms));
			diTmpTimeCounter:=0;
			iIncVelocity:=DINT_TO_INT(LREAL_TO_DINT(lrVelocity)/diTimeCounter);
			IF (iIncVelocity = 0) THEN
				IF (lrVelocity >= 0.0) THEN
					iIncVelocity:=1;
				END_IF;
				IF (lrVelocity < 0.0) THEN
					iIncVelocity:=-1;
				END_IF;
			END_IF;
			iStepMoveVelFB:=30;
		30:	iDataOut:=iDataOut + iIncVelocity;
			diTmpTimeCounter:=diTmpTimeCounter + 1;
			IF (diTmpTimeCounter >= diTimeCounter) THEN
				iDataOut:=LREAL_TO_INT(lrVelocity);
				iStepMoveVelFB:=900;
			END_IF;
			RETURN;
		900:	(* confirm reset *)
			xPowerOn:=TRUE;
			xPowerOff:=FALSE;
			T_Axis_DC.T_CtrleDCAxis.xPower:=TRUE;
			T_Axis_DC.T_CtrleDCAxis.xNotMoving:=FALSE;
			T_Axis_DC.T_CtrleDCAxis.xDone:=TRUE;
			T_Axis_DC.T_CtrleDCAxis.xErr:= FALSE;
			T_Axis_DC.T_CtrleDCAxis.udiErrorID:=16#0;
			(* init. variable *)
			xMoveVel:=FALSE;
		END_CASE;
	END_IF;

(* Send Parameter *)
	IF xSendAxisParameter THEN
		CASE iStepSendAxisParameterFB OF
		1:	TimerTimeOutFunction(IN:=FALSE);
			IF NOT(xWriteRegister) THEN
				IF (T_Axis_DC.T_ParamFileObj[iPtrAxisParameter].iBitValue = 16) THEN
					T_Axis_DC.T_CtrleDCAxis.iRegisterNr:=T_Axis_DC.T_ParamFileObj[iPtrAxisParameter].iRegisterNr;
					T_Axis_DC.T_CtrleDCAxis.iValueRegister:=LREAL_TO_INT(T_Axis_DC.T_ParamFileObj[iPtrAxisParameter].lrReal);
					xWriteRegister:=TRUE;
					iStepWriteRegister:=1;
					iPtrAxisParameter:=iPtrAxisParameter + 1;
				ELSE
					iStepSendAxisParameterFB:=10;
				END_IF;
			END_IF;
		10:	wDataToSend:=0;
			WHILE (T_Axis_DC.T_ParamFileObj[iPtrAxisParameter].iRegisterNr = 32) DO
				IF (T_Axis_DC.T_ParamFileObj[iPtrAxisParameter].lrReal <> 0) THEN
					wDataToSend:=wDataToSend OR REAL_TO_WORD(EXPT(2,T_Axis_DC.T_ParamFileObj[iPtrAxisParameter].iBitValue));
				END_IF;
				iPtrAxisParameter:=iPtrAxisParameter + 1;
			END_WHILE;
			iStepSendAxisParameterFB:=20;
		20:	T_Axis_DC.T_CtrleDCAxis.iRegisterNr:=32;
			T_Axis_DC.T_CtrleDCAxis.iValueRegister:=WORD_TO_INT(wDataToSend);
			xWriteRegister:=TRUE;
			iStepWriteRegister:=1;
			iStepSendAxisParameterFB:=30;
		30:	IF NOT(xWriteRegister) THEN
				iStepSendAxisParameterFB:=900;
			END_IF;
		900:	(* confirm reset *)
			T_Axis_DC.T_CtrleDCAxis.xDone:=TRUE;
			T_Axis_DC.T_CtrleDCAxis.xErr:= FALSE;
			T_Axis_DC.T_CtrleDCAxis.udiErrorID:=16#0;
			(* init. variable *)
			xSendAxisParameter:=FALSE;
		END_CASE;
	END_IF;

(* Write Register *)
	IF xWriteRegister THEN
		CASE iStepWriteRegister OF
		1:	TimerTimeOutFunction(IN:=FALSE);
			xTmpError:=FALSE;
			usiControlWord:=0;
			iDataOut:=16#0;
			iStepWriteRegister:=10;
		10:	IF (usiStatusWord = 16#0) OR (usiStatusWord = 16#20) THEN
			(* Leave Write protection for Register *)
				usiControlWord:=2#11111 + 2#11000000;
				iDataOut:=16#1235;
				iStepWriteRegister:=20;
			END_IF;
		20:	IF ((USINT_TO_BYTE(usiStatusWord) AND 2#10000000) = 2#10000000) THEN
				usiControlWord:=0;
				iDataOut:=16#0;
				iStepWriteRegister:=30;
			END_IF;
		30:	IF (usiStatusWord = 16#0) OR (usiStatusWord = 16#20) THEN
				(* send Data to write *)
				usiControlWord:=INT_TO_USINT(T_Axis_DC.T_CtrleDCAxis.iRegisterNr + 2#11000000);
				iDataOut:=T_Axis_DC.T_CtrleDCAxis.iValueRegister;
				iTmpDataOut:=iDataOut;
				iStepWriteRegister:=40;
			END_IF;
		(* wait for confirm *)
		40:	IF ((USINT_TO_BYTE(usiStatusWord) AND 2#10000000) = 2#10000000) THEN
				usiControlWord:=0;
				iDataOut:=16#0;
				iStepWriteRegister:=50;
			END_IF;
		50:	IF (usiStatusWord = 16#0) OR (usiStatusWord = 16#20) THEN
			(* check if data is writeted *)
				xReadRegister:=TRUE;
				iStepReadRegister:=1;
				iStepWriteRegister:=60;
			END_IF;
		60:	IF NOT(xReadRegister) THEN
				IF (T_Axis_DC.T_CtrleDCAxis.iValueRegister = iTmpDataOut) THEN
					iStepWriteRegister:=80;
				ELSE
					xTmpError:=TRUE;
					xResetAxis:=TRUE;
					iStepResetFB:=1;
					iStepWriteRegister:=70;
				END_IF;
			END_IF;
		70:	IF NOT(xResetAxis) THEN
				iStepWriteRegister:=80;
			END_IF;
		80:	usiControlWord:=0;
			iDataOut:=16#0;
			iStepWriteRegister:=90;
		90:	IF (usiStatusWord = 16#0) OR (usiStatusWord = 16#20) THEN
			(* Set Write protection for Register *)
				usiControlWord:=2#11111 + 2#11000000;
				iDataOut:=16#1111;
				iStepWriteRegister:=100;
			END_IF;
		100:	IF ((USINT_TO_BYTE(usiStatusWord) AND 2#10000000) = 2#10000000) THEN
				usiControlWord:=0;
				iDataOut:=16#0;
				iStepWriteRegister:=110;
			END_IF;
		110:	IF (usiStatusWord = 16#0) OR (usiStatusWord = 16#20) THEN
				IF NOT(xTmpError) THEN
					iStepWriteRegister:=900;
				ELSE
					iStepWriteRegister:=999;
				END_IF;
			END_IF;
		900:	(* confirm reset *)
			IF NOT(xInitAxis) AND NOT(xSendAxisParameter) THEN
				T_Axis_DC.T_CtrleDCAxis.xDone:=TRUE;
				T_Axis_DC.T_CtrleDCAxis.xErr:= FALSE;
				T_Axis_DC.T_CtrleDCAxis.udiErrorID:=16#0;
			END_IF;
			(* init. variable *)
			xWriteRegister:=FALSE;
		999:	(* Error stage *)
			T_Axis_DC.T_CtrleDCAxis.xDone:=FALSE;
			T_Axis_DC.T_CtrleDCAxis.xErr:= TRUE;
			T_Axis_DC.T_CtrleDCAxis.udiErrorID:=16#F600;	(* Can not set Data to Axiscontroller *)
			xWriteRegister:=FALSE;
			xInitAxis:=FALSE;
		END_CASE;
	END_IF;

(* Read Register *)
	IF xReadRegister THEN
		CASE iStepReadRegister OF
		1:	TimerTimeOutFunction(IN:=FALSE);
			xTmpError:=FALSE;
			usiControlWord:=0;
			iDataOut:=16#0;
			iStepReadRegister:=10;
		10:	IF (usiStatusWord = 16#0) OR (usiStatusWord = 16#20) THEN
			(* Leave Write protection for Register *)
				usiControlWord:=2#11111 + 2#11000000;
				iDataOut:=16#1235;
				iStepReadRegister:=20;
			END_IF;
		20:	IF ((USINT_TO_BYTE(usiStatusWord) AND 2#10000000) = 2#10000000) THEN
				usiControlWord:=0;
				iDataOut:=16#0;
				iStepReadRegister:=30;
			END_IF;
		30:	IF (usiStatusWord = 16#0) OR (usiStatusWord = 16#20) THEN
				usiControlWord:=INT_TO_USINT(T_Axis_DC.T_CtrleDCAxis.iRegisterNr + 2#10000000);
				iDataOut:=0;
				iStepReadRegister:=40;
			END_IF;
		40:	IF ((USINT_TO_WORD(usiStatusWord) AND 2#10000000) = 2#10000000) AND ((USINT_TO_WORD(usiStatusWord) AND 2#01000000) <> 2#01000000) THEN
				T_Axis_DC.T_CtrleDCAxis.iValueRegister:=iDataIn;
				iStepReadRegister:=50;
			END_IF;
			IF ((USINT_TO_WORD(usiStatusWord) AND 2#01000000) = 2#01000000) THEN
				T_Axis_DC.T_CtrleDCAxis.iValueRegister:=0;
				xTmpError:=TRUE;
				iStepReadRegister:=50;
			END_IF;
		50:	usiControlWord:=0;
			iDataOut:=16#0;
			iStepReadRegister:=60;
		60:	IF (usiStatusWord = 16#0) OR (usiStatusWord = 16#20) THEN
			(* Set Write protection for Register *)
				usiControlWord:=2#11111 + 2#11000000;
				iDataOut:=16#1111;
				iStepReadRegister:=70;
			END_IF;
		70:	IF ((USINT_TO_BYTE(usiStatusWord) AND 2#10000000) = 2#10000000) THEN
				usiControlWord:=0;
				iDataOut:=16#0;
				iStepReadRegister:=80;
			END_IF;
		80:	IF (usiStatusWord = 16#0) OR (usiStatusWord = 16#20) THEN
				IF NOT(xTmpError) THEN
					iStepReadRegister:=900;
				ELSE
					iStepReadRegister:=999;
				END_IF;
			END_IF;
		900:	(* confirm reset *)
			IF NOT(xWriteRegister) THEN
				T_Axis_DC.T_CtrleDCAxis.xDone:=TRUE;
				T_Axis_DC.T_CtrleDCAxis.xErr:= FALSE;
				T_Axis_DC.T_CtrleDCAxis.udiErrorID:=16#0;
			END_IF;
			(* init. variable *)
			xReadRegister:=FALSE;
		999:	(* Error stage *)
			T_Axis_DC.T_CtrleDCAxis.xDone:=FALSE;
			T_Axis_DC.T_CtrleDCAxis.xErr:= TRUE;
			T_Axis_DC.T_CtrleDCAxis.udiErrorID:=16#F700;	(* Can not read register from Axiscontroller *)
			(* init. variable *)
			xReadRegister:=FALSE;
			xWriteRegister:=FALSE;
		END_CASE;
	END_IF;
END_FUNCTION_BLOCK

(* POU FBDivers/FBConvertParaAxis, ST *)
FUNCTION_BLOCK FBConvertParaAxis
VAR_INPUT
	xStart:BOOL;
	iConversion:INT;
	sDeviceName:STRING(255);
END_VAR
VAR_IN_OUT
	T_Axis:ST_AXIS;
	T_Axis_DC : ST_DC_AXIS;
END_VAR
VAR_OUTPUT
	xDone:BOOL;
	xBusy:BOOL;
	xError:BOOL;
	diErrorNr:DINT;
END_VAR
VAR
(* trigger *)
	RisingEdgeStart:R_TRIG;
(* variable *)
	i: INT;
	iPosCarStart,iPosCarStop:INT;
	iStepConvertValueString:INT;
(* tmp variable *)
	sTmp:STRING(255);
	jj: INT;
END_VAR
(* wait start *)
	RisingEdgeStart(CLK:=xStart);
	IF RisingEdgeStart.Q THEN
	(* init. varaible *)
		iStepConvertValueString:=1;
		xDone:=FALSE;
	(*activ busy flag*)
		xBusy:=TRUE;
		xError:=FALSE;
		diErrorNr:=0;
	END_IF

(* test if activ *)
	IF NOT(xBusy) THEN
	(* exit FB *)
		RETURN;
	END_IF
	IF iConversion = 0 THEN
	(* conversion string to value *)
		i:=1;
		(* read string line-->Group or NodeId *)
		sTmp:=T_Axis.T_FileObj.sData[i];
		iPosCarStart:=FIND(sTmp,':=')+2;
		iPosCarStop:=FIND(sTmp,';');
		IF ((iPosCarStart - 2) = 0) OR (iPosCarStop = 0) OR (iPosCarStart >= iPosCarStop) THEN xBusy:=FALSE;	xDone:=FALSE; xError:=TRUE; diErrorNr:=16#F100;	(* Wrong Syntax from Axis File *) RETURN; END_IF;
		IF sDeviceName = 'Beckhoff' THEN
			T_Axis.T_Config_Gen.udiNC_TaskIdxGrp:=STRING_TO_UDINT(MID(sTmp,iPosCarStop-iPosCarStart,iPosCarStart));
			T_Axis.T_Config_Gen.udiNodeId:=0;
		END_IF;
		IF sDeviceName = 'Maxon' THEN
			T_Axis.T_Config_Gen.udiNC_TaskIdxGrp:=0;
			T_Axis.T_Config_Gen.udiNodeId:=STRING_TO_UDINT(MID(sTmp,iPosCarStop-iPosCarStart,iPosCarStart));
		END_IF;
		i:=i+1;
		(* read string line-->ADS NetID *)
		sTmp:=T_Axis.T_FileObj.sData[i];
		iPosCarStart:=FIND(sTmp,':=')+2;
		iPosCarStop:=FIND(sTmp,';');
		IF ((iPosCarStart - 2) = 0) OR (iPosCarStop = 0) OR (iPosCarStart >= iPosCarStop) THEN xBusy:=FALSE;	xDone:=FALSE; xError:=TRUE; diErrorNr:=16#F100;	(* Wrong Syntax from Axis File *) RETURN; END_IF;
		IF sDeviceName = 'Beckhoff' THEN
			T_Axis.T_Config_Gen.sServoNetId:=MID(sTmp,iPosCarStop-iPosCarStart,iPosCarStart);
			T_Axis.T_Config_Gen.sAmsNetId:='';
		END_IF;
		IF sDeviceName = 'Maxon' THEN
			T_Axis.T_Config_Gen.sServoNetId:='';
			T_Axis.T_Config_Gen.sAmsNetId:=MID(sTmp,iPosCarStop-iPosCarStart,iPosCarStart);
		END_IF;
		i:=i+1;
		(* read string line-->DeviceName *)
		sTmp:=T_Axis.T_FileObj.sData[i];
		iPosCarStart:=FIND(sTmp,':=')+2;
   		iPosCarStop:=FIND(sTmp,';');
		IF ((iPosCarStart - 2) = 0) OR (iPosCarStop = 0) OR (iPosCarStart >= iPosCarStop) THEN xBusy:=FALSE;	xDone:=FALSE; xError:=TRUE; diErrorNr:=16#F100;	(* Wrong Syntax from Axis File *) RETURN; END_IF;
		T_Axis.T_Config_Gen.sDeviceFileName:=MID(sTmp,iPosCarStop-iPosCarStart,iPosCarStart);
		i:=i+1;
		IF sDeviceName = 'Maxon' THEN
			(* read string line-->Scalefactor only for maxon motor *)
			sTmp:=T_Axis.T_FileObj.sData[i];
			iPosCarStart:=FIND(sTmp,':=')+2;
   			iPosCarStop:=FIND(sTmp,';');
			IF ((iPosCarStart - 2) = 0) OR (iPosCarStop = 0) OR (iPosCarStart >= iPosCarStop) THEN xBusy:=FALSE;	xDone:=FALSE; xError:=TRUE; diErrorNr:=16#F100;	(* Wrong Syntax from Axis File *) RETURN; END_IF;
			T_Axis.T_CtrleSingle.lrScaleFactor:=STRING_TO_REAL(MID(sTmp,iPosCarStop-iPosCarStart,iPosCarStart));
			i:=i+1;
			(* read string line-->NominalSpeed only for maxon motor *)
			sTmp:=T_Axis.T_FileObj.sData[i];
			iPosCarStart:=FIND(sTmp,':=')+2;
   			iPosCarStop:=FIND(sTmp,';');
			IF ((iPosCarStart - 2) = 0) OR (iPosCarStop = 0) OR (iPosCarStart >= iPosCarStop) THEN xBusy:=FALSE;	xDone:=FALSE; xError:=TRUE; diErrorNr:=16#F100;	(* Wrong Syntax from Axis File *) RETURN; END_IF;
			T_Axis.T_CtrleSingle.rNominalSpeed:=STRING_TO_REAL(MID(sTmp,iPosCarStop-iPosCarStart,iPosCarStart));
			i:=i+1;
		END_IF;
		IF sDeviceName = 'Beckhoff' THEN
			(* read string line-->Quickstop ramp deceleration *)
			sTmp:=T_Axis.T_FileObj.sData[i];
			iPosCarStart:=FIND(sTmp,':=')+2;
	   		iPosCarStop:=FIND(sTmp,';');
			IF ((iPosCarStart - 2) = 0) OR (iPosCarStop = 0) OR (iPosCarStart >= iPosCarStop) THEN xBusy:=FALSE;	xDone:=FALSE; xError:=TRUE; diErrorNr:=16#F100;	(* Wrong Syntax from Axis File *) RETURN; END_IF;
			T_Axis.T_Config_Setting.rHCRampDeceleration:=STRING_TO_REAL(MID(sTmp,iPosCarStop-iPosCarStart,iPosCarStart));
			i:=i+1;
			(* read string line-->Quickstop ramp jerk *)
			sTmp:=T_Axis.T_FileObj.sData[i];
			iPosCarStart:=FIND(sTmp,':=')+2;
	   		iPosCarStop:=FIND(sTmp,';');
			IF ((iPosCarStart - 2) = 0) OR (iPosCarStop = 0) OR (iPosCarStart >= iPosCarStop) THEN xBusy:=FALSE;	xDone:=FALSE; xError:=TRUE; diErrorNr:=16#F100;	(* Wrong Syntax from Axis File *) RETURN; END_IF;
			T_Axis.T_Config_Setting.rHCRampJerk:=STRING_TO_REAL(MID(sTmp,iPosCarStop-iPosCarStart,iPosCarStart));
			i:=i+1;
		END_IF;
		jj:=1;
		(* read string lines *)
		WHILE T_Axis.T_FileObj.sData[i] <> '' DO
			sTmp:=T_Axis.T_FileObj.sData[i];
			(* index group *)
			iPosCarStart:=FIND(sTmp,':=')+2;
			iPosCarStop:=FIND(sTmp,';');
			IF ((iPosCarStart - 2) = 0) OR (iPosCarStop = 0) OR (iPosCarStart >= iPosCarStop) THEN xBusy:=FALSE;	xDone:=FALSE; xError:=TRUE; diErrorNr:=16#F100;	(* Wrong Syntax from Axis File *) RETURN; END_IF;
			T_Axis.T_ParamFileObj[jj].udiIdxGroup:=	STRING_TO_UDINT(MID(sTmp,iPosCarStop-iPosCarStart,iPosCarStart))
											+ T_Axis.T_Config_Gen.udiNC_TaskIdxGrp;
			sTmp:=MID(sTmp,LEN(sTmp)-iPosCarStop, iPosCarStop+1);
			(* index offset *)
			iPosCarStart:=FIND(sTmp,':=')+2;
			iPosCarStop:=FIND(sTmp,';');
			IF ((iPosCarStart - 2) = 0) OR (iPosCarStop = 0) OR (iPosCarStart >= iPosCarStop) THEN xBusy:=FALSE;	xDone:=FALSE; xError:=TRUE; diErrorNr:=16#F100;	(* Wrong Syntax from Axis File *) RETURN; END_IF;
			T_Axis.T_ParamFileObj[jj].udiIndexOffset:=STRING_TO_UDINT(MID(sTmp,iPosCarStop-iPosCarStart,iPosCarStart));
			sTmp:=MID(sTmp,LEN(sTmp)-iPosCarStop, iPosCarStop+1);
			(* length value *)
			iPosCarStart:=FIND(sTmp,':=')+2;
			iPosCarStop:=FIND(sTmp,';');
			IF ((iPosCarStart - 2) = 0) OR (iPosCarStop = 0) OR (iPosCarStart >= iPosCarStop) THEN xBusy:=FALSE;	xDone:=FALSE; xError:=TRUE; diErrorNr:=16#F100;	(* Wrong Syntax from Axis File *) RETURN; END_IF;
			T_Axis.T_ParamFileObj[jj].udiLength:=STRING_TO_UDINT(MID(sTmp,iPosCarStop-iPosCarStart,iPosCarStart));
			sTmp:=MID(sTmp,LEN(sTmp)-iPosCarStop, iPosCarStop+1);
			(* value*)
			iPosCarStart:=FIND(sTmp,':=')+2;
			iPosCarStop:=FIND(sTmp,';');
			IF ((iPosCarStart - 2) = 0) OR (iPosCarStop = 0) OR (iPosCarStart >= iPosCarStop) THEN xBusy:=FALSE;	xDone:=FALSE; xError:=TRUE; diErrorNr:=16#F100;	(* Wrong Syntax from Axis File *) RETURN; END_IF;
			T_Axis.T_ParamFileObj[jj].lrReal:=STRING_TO_REAL(MID(sTmp,iPosCarStop-iPosCarStart,iPosCarStart));
			(* init existing line, erase text *)
			iPosCarStop:=FIND(T_Axis.T_FileObj.sData[i],'(');
			T_Axis.T_FileObj.sData[i]:=MID(T_Axis.T_FileObj.sData[i],iPosCarStop-1,1);
			(* next line *)
			i:=i+1;
			jj:=jj+1;
		END_WHILE
		(* init. next *)
		T_Axis.T_ParamFileObj[jj].udiIdxGroup:=0;
		T_Axis.T_ParamFileObj[jj].udiIndexOffset:=0;
		T_Axis.T_ParamFileObj[jj].udiLength:=0;
		T_Axis.T_ParamFileObj[jj].lrReal:=0;

	(* Init. NC parameter *)
		i:=1;
		(* Beckhoff *)
		IF sDeviceName = 'Beckhoff' THEN
			(*copy parameter value *)
			WHILE T_Axis.T_ParamFileObj[i].udiIdxGroup <> 0 DO
				CASE (T_Axis.T_ParamFileObj[i].udiIdxGroup - T_Axis.T_Config_Gen.udiNC_TaskIdxGrp) OF
				16#4000:	CASE T_Axis.T_ParamFileObj[i].udiIndexOffset OF
						(* Calibration velocity forward *)
						16#6:	T_Axis.T_Config_ObjFileValue.lrCalVelocityForward:=T_Axis.T_ParamFileObj[i].lrReal;
						(* Calibration velocity backward *)
						16#7:	T_Axis.T_Config_ObjFileValue.lrCalVelocityBackward:=T_Axis.T_ParamFileObj[i].lrReal;
						(* Maximum velocity *)
						16#27:	T_Axis.T_Config_ObjFileValue.lrMaxVelocity:=T_Axis.T_ParamFileObj[i].lrReal;
						(* Acceleration *)
						16#101:	T_Axis.T_Config_ObjFileValue.lrAcceleration:=T_Axis.T_ParamFileObj[i].lrReal;
						(* Decceleration *)
						16#102:	T_Axis.T_Config_ObjFileValue.lrDecceleration:=T_Axis.T_ParamFileObj[i].lrReal;
						(* Jerk *)
						16#103:	T_Axis.T_Config_ObjFileValue.lrJerk:=T_Axis.T_ParamFileObj[i].lrReal;
						END_CASE
				16#5000:	CASE T_Axis.T_ParamFileObj[i].udiIndexOffset OF
						(* Encoder scaling factor *)
						16#6:	T_Axis.T_Config_ObjFileValue.lrScaleFactor:=T_Axis.T_ParamFileObj[i].lrReal;
						(* SW limit negativ On/Off *)
						16#B:	T_Axis.T_Config_ObjFileValue.xSWLimitNeg:=REAL_TO_BOOL(T_Axis.T_ParamFileObj[i].lrReal);
						(* SW limit positiv On/Off *)
						16#C:	T_Axis.T_Config_ObjFileValue.xSWLimitPos:=REAL_TO_BOOL(T_Axis.T_ParamFileObj[i].lrReal);
						(* SW limit negativ value *)
						16#D:	T_Axis.T_Config_ObjFileValue.lrSWLimitNeg:=T_Axis.T_ParamFileObj[i].lrReal;
						(* SW limit position value *)
						16#E:	T_Axis.T_Config_ObjFileValue.lrSWLimitPos:=T_Axis.T_ParamFileObj[i].lrReal;
						END_CASE
				16#6000:;
				16#7000:;
				END_CASE
				(* next parameter *)
				i:=i+1;
			END_WHILE
		END_IF

		(* Maxon *)
		IF sDeviceName = 'Maxon' THEN
			(*copy parameter value *)
			WHILE T_Axis.T_ParamFileObj[i].udiIdxGroup <> 0 DO
				CASE T_Axis.T_ParamFileObj[i].udiIdxGroup  OF
				16#6083:	CASE T_Axis.T_ParamFileObj[i].udiIndexOffset OF
						(* Acceleration *)
						16#0:	T_Axis.T_Config_ObjFileValue.lrAcceleration:=T_Axis.T_ParamFileObj[i].lrReal;
						END_CASE
				16#6084:	CASE T_Axis.T_ParamFileObj[i].udiIndexOffset OF
						(* Decceleration *)
						16#0:	T_Axis.T_Config_ObjFileValue.lrDecceleration:=T_Axis.T_ParamFileObj[i].lrReal;
						END_CASE
				END_CASE
				(* next parameter *)
				i:=i+1;
			END_WHILE
		END_IF
		(* set flag done *)
		xBusy:=FALSE;
		xDone:=TRUE;
	END_IF;
	IF iConversion = 1 THEN
	(* conversion string to value *)
		i:=1;
		(* read string line-->Group or NodeId *)
		sTmp:=T_Axis_DC.T_FileObj.sData[i];
		iPosCarStart:=FIND(sTmp,':=')+2;
		iPosCarStop:=FIND(sTmp,';');
		IF ((iPosCarStart - 2) = 0) OR (iPosCarStop = 0) OR (iPosCarStart >= iPosCarStop) THEN xBusy:=FALSE;	xDone:=FALSE; xError:=TRUE; diErrorNr:=16#F100;	(* Wrong Syntax from Axis File *) RETURN; END_IF;
		T_Axis_DC.T_Config_Gen.udiNodeId:=STRING_TO_UDINT(MID(sTmp,iPosCarStop-iPosCarStart,iPosCarStart));
		i:=i+1;
		(* read string line-->DeviceName *)
		sTmp:=T_Axis_DC.T_FileObj.sData[i];
		iPosCarStart:=FIND(sTmp,':=')+2;
   		iPosCarStop:=FIND(sTmp,';');
		IF ((iPosCarStart - 2) = 0) OR (iPosCarStop = 0) OR (iPosCarStart >= iPosCarStop) THEN xBusy:=FALSE;	xDone:=FALSE; xError:=TRUE; diErrorNr:=16#F100;	(* Wrong Syntax from Axis File *) RETURN; END_IF;
		T_Axis_DC.T_Config_Gen.sDeviceFileName:=MID(sTmp,iPosCarStop-iPosCarStart,iPosCarStart);
		i:=i+1;
		(* read string line-->Scalefactor *)
		sTmp:=T_Axis_DC.T_FileObj.sData[i];
		iPosCarStart:=FIND(sTmp,':=')+2;
		iPosCarStop:=FIND(sTmp,';');
		IF ((iPosCarStart - 2) = 0) OR (iPosCarStop = 0) OR (iPosCarStart >= iPosCarStop) THEN xBusy:=FALSE;	xDone:=FALSE; xError:=TRUE; diErrorNr:=16#F100;	(* Wrong Syntax from Axis File *) RETURN; END_IF;
		T_Axis_DC.T_Config_Gen.lrScaleFactor:=STRING_TO_LREAL(MID(sTmp,iPosCarStop-iPosCarStart,iPosCarStart));
		i:=i+1;
		(* read string line-->Initfactor *)
		sTmp:=T_Axis_DC.T_FileObj.sData[i];
		iPosCarStart:=FIND(sTmp,':=')+2;
		iPosCarStop:=FIND(sTmp,';');
		IF ((iPosCarStart - 2) = 0) OR (iPosCarStop = 0) OR (iPosCarStart >= iPosCarStop) THEN xBusy:=FALSE;	xDone:=FALSE; xError:=TRUE; diErrorNr:=16#F100;	(* Wrong Syntax from Axis File *) RETURN; END_IF;
		T_Axis_DC.T_Config_Gen.lrInitFactor:=STRING_TO_LREAL(MID(sTmp,iPosCarStop-iPosCarStart,iPosCarStart));
		i:=i+1;
		(* read string lines *)
		WHILE T_Axis_DC.T_FileObj.sData[i] <> '' DO
			sTmp:=T_Axis_DC.T_FileObj.sData[i];
			(* index Register number *)
			iPosCarStart:=FIND(sTmp,':=')+2;
			iPosCarStop:=FIND(sTmp,';');
			IF ((iPosCarStart - 2) = 0) OR (iPosCarStop = 0) OR (iPosCarStart >= iPosCarStop) THEN xBusy:=FALSE;	xDone:=FALSE; xError:=TRUE; diErrorNr:=16#F100;	(* Wrong Syntax from Axis File *) RETURN; END_IF;
			T_Axis_DC.T_ParamFileObj[i - 4].iRegisterNr :=	STRING_TO_INT(MID(sTmp,iPosCarStop-iPosCarStart,iPosCarStart));
			sTmp:=MID(sTmp,LEN(sTmp)-iPosCarStop, iPosCarStop+1);
			(* index bit value *)
			iPosCarStart:=FIND(sTmp,':=')+2;
			iPosCarStop:=FIND(sTmp,';');
			IF ((iPosCarStart - 2) = 0) OR (iPosCarStop = 0) OR (iPosCarStart >= iPosCarStop) THEN xBusy:=FALSE;	xDone:=FALSE; xError:=TRUE; diErrorNr:=16#F100;	(* Wrong Syntax from Axis File *) RETURN; END_IF;
			T_Axis_DC.T_ParamFileObj[i - 4].iBitValue:=STRING_TO_INT(MID(sTmp,iPosCarStop-iPosCarStart,iPosCarStart));
			sTmp:=MID(sTmp,LEN(sTmp)-iPosCarStop, iPosCarStop+1);
			(* value*)
			iPosCarStart:=FIND(sTmp,':=')+2;
			iPosCarStop:=FIND(sTmp,';');
			IF ((iPosCarStart - 2) = 0) OR (iPosCarStop = 0) OR (iPosCarStart >= iPosCarStop) THEN xBusy:=FALSE;	xDone:=FALSE; xError:=TRUE; diErrorNr:=16#F100;	(* Wrong Syntax from Axis File *) RETURN; END_IF;
			T_Axis_DC.T_ParamFileObj[i - 4].lrReal:=STRING_TO_REAL(MID(sTmp,iPosCarStop-iPosCarStart,iPosCarStart));
			(* init existing line, erase text *)
			iPosCarStop:=FIND(T_Axis_DC.T_FileObj.sData[i],'(');
			T_Axis_DC.T_FileObj.sData[i]:=MID(T_Axis_DC.T_FileObj.sData[i],iPosCarStop-1,1);
			(* next line *)
			i:=i+1;
		END_WHILE
		(* init. next *)
		T_Axis_DC.T_ParamFileObj[i - 4].iRegisterNr:=0;
		T_Axis_DC.T_ParamFileObj[i - 4].iBitValue:=0;
		T_Axis_DC.T_ParamFileObj[i - 4].lrReal:=0;
		(* Init Parameter *)
		i:=1;
		IF sDeviceName = 'MaxonDC' THEN
			(*copy parameter value *)
			WHILE T_Axis_DC.T_ParamFileObj[i].iRegisterNr <> 0 DO
				CASE T_Axis_DC.T_ParamFileObj[i].iRegisterNr OF
				36:	T_Axis_DC.T_Config_ObjFileValue.diMaxMotorCurrent:=LREAL_TO_DINT(T_Axis_DC.T_ParamFileObj[i].lrReal);
				37:	T_Axis_DC.T_Config_ObjFileValue.diNominalMotorCurrent:=LREAL_TO_DINT(T_Axis_DC.T_ParamFileObj[i].lrReal);
				40:	T_Axis_DC.T_Config_ObjFileValue.diMotorResistor:=LREAL_TO_DINT(T_Axis_DC.T_ParamFileObj[i].lrReal);
				42:	T_Axis_DC.T_Config_ObjFileValue.diKpSpeedControl:=LREAL_TO_DINT(T_Axis_DC.T_ParamFileObj[i].lrReal);
				45:	T_Axis_DC.T_Config_ObjFileValue.diTnCurrentControl:=LREAL_TO_DINT(T_Axis_DC.T_ParamFileObj[i].lrReal);
				38:	T_Axis_DC.T_Config_ObjFileValue.diMaxTorqueMotor:=LREAL_TO_DINT(T_Axis_DC.T_ParamFileObj[i].lrReal);
				32:	CASE T_Axis_DC.T_ParamFileObj[i].iBitValue OF
					15:	IF (T_Axis_DC.T_ParamFileObj[i].lrReal = 0) THEN T_Axis_DC.T_Config_ObjFileValue.xSpeedControlAcitv:=TRUE; END_IF;
						IF (T_Axis_DC.T_ParamFileObj[i].lrReal = 1) THEN T_Axis_DC.T_Config_ObjFileValue.xSpeedControlAcitv:=FALSE; END_IF;
					14:	IF (T_Axis_DC.T_ParamFileObj[i].lrReal = 0) THEN T_Axis_DC.T_Config_ObjFileValue.xCurrentControlAcitv:=TRUE; END_IF;
						IF (T_Axis_DC.T_ParamFileObj[i].lrReal = 1) THEN T_Axis_DC.T_Config_ObjFileValue.xCurrentControlAcitv:=FALSE; END_IF;
					13:	IF (T_Axis_DC.T_ParamFileObj[i].lrReal = 0) THEN T_Axis_DC.T_Config_ObjFileValue.xWinCurrentControlActiv:=TRUE; END_IF;
						IF (T_Axis_DC.T_ParamFileObj[i].lrReal = 1) THEN T_Axis_DC.T_Config_ObjFileValue.xWinCurrentControlActiv:=FALSE; END_IF;
					09:	IF (T_Axis_DC.T_ParamFileObj[i].lrReal = 0) THEN T_Axis_DC.T_Config_ObjFileValue.xTorqueControlAcitv:=FALSE; END_IF;
						IF (T_Axis_DC.T_ParamFileObj[i].lrReal = 1) THEN T_Axis_DC.T_Config_ObjFileValue.xTorqueControlAcitv:=TRUE; END_IF;
					10:	IF (T_Axis_DC.T_ParamFileObj[i].lrReal = 0) THEN T_Axis_DC.T_Config_ObjFileValue.xOverVoltageActiv:=FALSE; END_IF;
						IF (T_Axis_DC.T_ParamFileObj[i].lrReal = 1) THEN T_Axis_DC.T_Config_ObjFileValue.xOverVoltageActiv:=TRUE; END_IF;
					END_CASE;
				END_CASE;
				i:=i+1;
			END_WHILE;
		END_IF;
		(* set flag done *)
		xBusy:=FALSE;
		xDone:=TRUE;
	END_IF;
END_FUNCTION_BLOCK

(* POU FB_HARDWARE/FBHW_CYL_ANALOG, ST *)
FUNCTION_BLOCK FBHW_CYL_ANALOG
VAR_INPUT
	xCtrlePosOn:BOOL;
	xCtrlePosOff:BOOL;
	iAnalogIn:INT;
END_VAR
VAR_OUTPUT
	iAnalogOut:INT;
END_VAR
VAR_IN_OUT
	T_Cylinder:ST_CYLINDER;
END_VAR
VAR
(* variable *)
	xConfirmResetFB: BOOL;
	iStep:INT;
(* timer *)
	TimerOn:TON;
	TimerOff:TON;
	TimerPreOn:TON;
	TimerPreOff:TON;
	TimerOut:TON;
	TimerActiv: TON;
(* trigger *)
	RisingEdgeExecute:R_TRIG;
	RisingEdgeReset:R_TRIG;
	RisingEdgeActiv:R_TRIG;
	FallingEdgeActiv:F_TRIG;
	xActiveRampFct: BOOL;
	FBCylAnalogFunction: FB_CylAnalogFunction;
	xStartRampFct: BOOL;
	iTmpAnalogIn: INT;
	xResetRampFct: BOOL;
	TimerAfterSensor: TON;
END_VAR
(* if function bloc set activ then Analog state will be transfered *)
	RisingEdgeActiv(CLK:=T_Cylinder.T_CtrleCyl.xFBActiv);
	FallingEdgeActiv(CLK:=T_Cylinder.T_CtrleCyl.xFBActiv);
	IF RisingEdgeActiv.Q OR FallingEdgeActiv.Q THEN
	(* set Analog Out = In on the rising edge from the activ signal *)
		iAnalogOut:=0;
		T_Cylinder.T_CtrleCyl.T_Analog.xActiv:= FALSE;
	END_IF

(* if bloc disable if activ signal is inactiv *)
	IF T_Cylinder.T_CtrleCyl.xFBActiv THEN
	(* copy control position state *)
		T_Cylinder.T_CtrleCyl.xStatePosOn:=xCtrlePosOn;
		T_Cylinder.T_CtrleCyl.xStatePosOff:=xCtrlePosOff;
	ELSE
	(* exit FB *)
		RETURN;
	END_IF

(* wait for reseting *)
	RisingEdgeReset(CLK:=T_Cylinder.T_CtrleCyl.xReset);
	IF RisingEdgeReset.Q THEN
		(* Init. timer *)
		TimerOn(IN:=TRUE,PT:=T#1ms);
		TimerOff(IN:=TRUE,PT:=T#1ms);
		TimerPreOn(IN:=TRUE,PT:=T#1ms);
		TimerPreOff(IN:=TRUE,PT:=T#1ms);
		TimerOut(IN:=TRUE,PT:=T#1ms);
	(* Init. variable *)
		iStep:=0;
	(* Init. structure *)
		T_Cylinder.T_CtrleCyl.iFunction:=0;
		T_Cylinder.T_CtrleCyl.T_Analog.xActiv:=FALSE;
		IF NOT(T_Cylinder.T_Config.xActivState) THEN
			iAnalogOut:=iAnalogIn;
		ELSE
			iAnalogOut:=0;
		END_IF;
		T_Cylinder.T_CtrleCyl.xDone:=FALSE;
		T_Cylinder.T_CtrleCyl.xErr:=FALSE;
		T_Cylinder.T_CtrleCyl.udiErrorID:=16#0;
		xActiveRampFct:=xStartRampFct:=FALSE;
		xResetRampFct:=TRUE;
		FBCylAnalogFunction(	xStart:= xStartRampFct,
							xReset:=xResetRampFct);
	(* confirm reset *)
		xConfirmResetFB:=TRUE;
	(* exit function *)
		RETURN;
	ELSE
		IF xConfirmResetFB THEN
		(* confirm reset FB *)
			T_Cylinder.T_CtrleCyl.xDone:=TRUE;
			T_Cylinder.T_CtrleCyl.xErr:=FALSE;
			T_Cylinder.T_CtrleCyl.udiErrorID:=16#0;
			(* reset variable *)
			xConfirmResetFB:=FALSE;
		END_IF
	END_IF

(* if bloc disable if activ signal is inactiv *)
	IF NOT(T_Cylinder.T_CtrleCyl.xFBActiv) THEN
		RETURN;
	END_IF

(* check active state of the servo valve *)
IF (iAnalogOut <> 0) THEN
	T_Cylinder.T_CtrleCyl.T_Analog.xActiv:=TRUE;
ELSE
	T_Cylinder.T_CtrleCyl.T_Analog.xActiv:=FALSE;
END_IF;

(* wait for execute *)
	RisingEdgeExecute(CLK:=T_Cylinder.T_CtrleCyl.xExecute);
	IF RisingEdgeExecute.Q THEN
		IF NOT(T_Cylinder.T_CtrleCyl.xDone) AND NOT(T_Cylinder.T_CtrleCyl.xErr) THEN
		(* can execute function if both signal are disable *)
			RETURN;
		END_IF
		CASE T_Cylinder.T_CtrleCyl.iFunction OF
		(* disable *)
		1:	iStep:=11;
		(* Activ without sensor position ctrle *)
		2:	iStep:=1;
		(* set value Analog Out = Analog In *)
		4:	iStep:=21;
		(* inverse cylinder state *)
		51:	iStep:=51;
		ELSE
			(* function not implemented *)
			iStep:=0;
			T_Cylinder.T_CtrleCyl.xDone:=FALSE;
			T_Cylinder.T_CtrleCyl.xErr:=TRUE;
			T_Cylinder.T_CtrleCyl.udiErrorID:=16#F000;
			(* exit FB *)
			RETURN;
		END_CASE
		(* Init. variable *)
		T_Cylinder.T_CtrleCyl.xDone:=FALSE;
		T_Cylinder.T_CtrleCyl.xErr:=FALSE;
		T_Cylinder.T_CtrleCyl.udiErrorID:=16#0;
		(* exit FB *)
		RETURN;
	END_IF

(* Timer activ *)
	TimerOn(IN:=TRUE,PT:=T_Cylinder.T_Config.tDelayOn);
	TimerOff(IN:=TRUE,PT:=T_Cylinder.T_Config.tDelayOff);
	TimerPreOn(IN:=TRUE,PT:=T_Cylinder.T_Config.tDelayPreOn);
	TimerPreOff(IN:=TRUE,PT:=T_Cylinder.T_Config.tDelayPreOff);
	TimerOut(IN:=TRUE,PT:=T_Cylinder.T_Config.tTimeOut);
	TimerActiv(IN:=TRUE,PT:=T_Cylinder.T_CtrleCyl.T_Analog.tDelayActiv);
	TimerAfterSensor(IN:=TRUE,PT:=T_Cylinder.T_CtrleCyl.T_Analog.tDelayAfterSensor);

(* waiting for activ *)
	CASE iStep OF
	(* process timer On *)
	1:	IF (T_Cylinder.T_Config.tDelayPreOn = T#0s) THEN
			TimerOn(IN:=FALSE);
			IF (iAnalogIn <> iAnalogOut) AND T_Cylinder.T_Config.xActivState THEN
				iTmpAnalogIn:=iAnalogIn;
				xActiveRampFct:=TRUE;
				iStep:=2;
			ELSIF (iAnalogOut <> 0) AND NOT(T_Cylinder.T_Config.xActivState) THEN
				iTmpAnalogIn:=0;
				xActiveRampFct:=TRUE;
				iStep:=2;
			ELSE
				iStep:=3;
			END_IF;
		ELSE
			TimerPreOn(IN:=FALSE);
			iStep:=4;
		END_IF;
	(* wait for timer On *)
	2:	IF TimerOn.Q AND NOT(xActiveRampFct) THEN
			iStep:=3;
			TimerOut(IN:=FALSE);
		END_IF
	(* control position activ *)
	3:	IF T_Cylinder.T_Config.xCtrlePosOn THEN
		(* position ctrle activ *)
			IF TimerOut.Q THEN
			(* timerout done, activ error cylinder has not activ position reached *)
				iStep:=999;
			ELSE
				IF xCtrlePosOn THEN
				(* Activ position reached, activ confirmation *)
					iStep:=80;
				END_IF
			END_IF
		ELSE
		(* no position ctrle, activ confirm *)
			iStep:=90;
		END_IF
	(* wait for timer Pre On *)
	4:	IF TimerPreOn.Q THEN
			T_Cylinder.T_Config.tDelayPreOn:=T#0s;
			iStep:=1;
		END_IF
	(* process timer Off *)
	11:	IF (T_Cylinder.T_Config.tDelayPreOff = T#0s) THEN
			TimerOff(IN:=FALSE);
			IF (iAnalogIn <> iAnalogOut) AND NOT(T_Cylinder.T_Config.xActivState) THEN
				iTmpAnalogIn:=iAnalogIn;
				xActiveRampFct:=TRUE;
				iStep:=12;
			ELSIF (iAnalogOut <> 0) AND T_Cylinder.T_Config.xActivState THEN
				iTmpAnalogIn:=0;
				xActiveRampFct:=TRUE;
				iStep:=12;
			ELSE
				iStep:=12;
			END_IF;
		ELSE
			TimerPreOff(IN:=FALSE);
			iStep:=14;
		END_IF;
	(* wait for timer Off *)
	12:	IF TimerOff.Q AND NOT(xActiveRampFct) THEN
			iStep:=13;
			TimerOut(IN:=FALSE);
		END_IF
	(* control position inactiv *)
	13:	IF T_Cylinder.T_Config.xCtrlePosOff THEN
		(* control position activ *)
			IF TimerOut.Q THEN
			(* timerout done, activ error 'cylinder has not inactiv position reached' *)
				iStep:=998;
			ELSE
				IF xCtrlePosOff THEN
				(* inactiv position reached, activ confirmation *)
					iStep:=85;
				END_IF
			END_IF
		ELSE
		(* no control position activ, activ confirmation *)
			iStep:=99;
		END_IF
	(* wait for timer Pre Off *)
	14:	IF TimerPreOff.Q THEN
			T_Cylinder.T_Config.tDelayPreOff:=T#0s;
			iStep:=11;
		END_IF
	(* set value Analog Out = Analog In *)
	21:	iTmpAnalogIn:=iAnalogIn;
		xActiveRampFct:=TRUE;
		iStep:=99;
	(* inverse cylinder state *)
	51:	IF (T_Cylinder.T_CtrleCyl.T_Analog.xActiv AND T_Cylinder.T_Config.xActivState) OR (NOT(T_Cylinder.T_CtrleCyl.T_Analog.xActiv) AND NOT(T_Cylinder.T_Config.xActivState)) THEN
			iTmpAnalogIn:=0;
			xActiveRampFct:=TRUE;
		END_IF;
		IF (T_Cylinder.T_CtrleCyl.T_Analog.xActiv AND NOT(T_Cylinder.T_Config.xActivState)) OR (NOT(T_Cylinder.T_CtrleCyl.T_Analog.xActiv) AND T_Cylinder.T_Config.xActivState) THEN
			iTmpAnalogIn:=iAnalogIn;
			xActiveRampFct:=TRUE;
		END_IF;
		iStep:=99;
	80:	IF (T_Cylinder.T_CtrleCyl.T_Analog.tDelayAfterSensor <> T#0s) THEN
			TimerAfterSensor(IN:=FALSE);
			iStep:=81;
		ELSE
			iStep:=90;
		END_IF;
	(* wait for time after sensor *)
	81:	IF TimerAfterSensor.Q THEN
			iStep:=90;
		END_IF
	85:	IF (T_Cylinder.T_CtrleCyl.T_Analog.tDelayAfterSensor <> T#0s) THEN
			TimerAfterSensor(IN:=FALSE);
			iStep:=86;
		ELSE
			iStep:=99;
		END_IF;
	(* wait for time after sensor *)
	86:	IF TimerAfterSensor.Q THEN
			iStep:=99;
		END_IF
	(* test if delay activ *)
	90:	IF T_Cylinder.T_CtrleCyl.T_Analog.tDelayActiv <> T#0s THEN
			TimerActiv(IN:=FALSE);
			iStep:=98;
		ELSE
			iStep:=99;
		END_IF
	(* wait for time delay activ *)
	98:	IF TimerActiv.Q THEN
		(* activ time is over, set variable off *)
			IF NOT(T_Cylinder.T_Config.xActivState) THEN
				iTmpAnalogIn:=iAnalogIn;
				xActiveRampFct:=TRUE;
			ELSE
				iTmpAnalogIn:=0;
				xActiveRampFct:=TRUE;
			END_IF;
			iStep:=99;
		END_IF
	(* process end *)
	99:	IF NOT(xActiveRampFct) THEN
			T_Cylinder.T_CtrleCyl.xDone:=TRUE;
			T_Cylinder.T_CtrleCyl.xErr:=FALSE;
			T_Cylinder.T_CtrleCyl.udiErrorID:=16#0;
		END_IF;
	(* error, cylinder not in inactiv position *)
	998:	T_Cylinder.T_CtrleCyl.xDone:=FALSE;
		T_Cylinder.T_CtrleCyl.xErr:=TRUE;
		T_Cylinder.T_CtrleCyl.udiErrorID:=16#F202;
	(* error, cylinder not in activ position *)
	999:	T_Cylinder.T_CtrleCyl.xDone:=FALSE;
		T_Cylinder.T_CtrleCyl.xErr:=TRUE;
		T_Cylinder.T_CtrleCyl.udiErrorID:=16#F201;
	END_CASE
(* Set Analog Output with or without Ramp *)
	IF xActiveRampFct THEN
		xStartRampFct:=TRUE;
		FBCylAnalogFunction(	iRampFctOn:= T_Cylinder.T_CtrleCyl.T_Analog.iRampFctOn,
							iRampFctOff:= T_Cylinder.T_CtrleCyl.T_Analog.iRampFctOff,
							rSetOutput:= INT_TO_REAL(iTmpAnalogIn),
							rDeltaOutput:= T_Cylinder.T_CtrleCyl.T_Analog.rStepValue,
							rTau:= 0.0,
							rActualOutput:=INT_TO_REAL(iAnalogOut),
							xStart:= xStartRampFct,
							xReset:=xResetRampFct);
		iAnalogOut:=REAL_TO_INT(FBCylAnalogFunction.rOutput);
		T_Cylinder.T_CtrleCyl.T_Analog.tTimeActivOn:=FBCylAnalogFunction.tOutputTimeOn;
		T_Cylinder.T_CtrleCyl.T_Analog.tTimeActivOff:=FBCylAnalogFunction.tOutputTimeOff;
		IF FBCylAnalogFunction.xEnd THEN
			xActiveRampFct:=xStartRampFct:=FALSE;
			T_Cylinder.T_CtrleCyl.T_Analog.rStepValue:=0.0;
		END_IF;
	END_IF;
END_FUNCTION_BLOCK

